# B&R Automation Studio project OpcUaSample410_BrbLibUa103 (part 18)

#### ClientST.st - Implementation code
```iecst
PROGRAM _INIT
	// Initialisierung des Tasks
	brsmemset(ADR(ClientVarsSubscription), 0, SIZEOF(ClientVarsSubscription)); // Auf diese Variablen werden die vom Server geschickten Werte geschrieben
	fbTrigger.PT := T#1s;
	brsmemset(ADR(ClientVarsRead), 0, SIZEOF(ClientVarsRead)); // Auf diese Variablen werden die vom Server gelesenen Werte geschrieben
	brsmemset(ADR(ReceivedEvent), 0, SIZEOF(ReceivedEvent)); // Auf diese Variablen werden die vom Server empfangenen Event-Felder geschrieben

	// Initialisierung der Schrittkette
	Step.eStepNr := eSTEP_INIT;
	bStartClient := 1; // Der Client startet erst, wenn auf 1. Kann zum Debugging auf 0 gesetzt werden.

	// Vorbesetzen der Konfiguration
	ClientCfg.Connection.sServerEndpointUrl := 'opc.tcp://localhost:4840';
	//ClientCfg.Connection.sServerEndpointUrl := 'opc.tcp://192.168.178.37:4840'; // Nur zum Test
	ClientCfg.Connection.UserIdentityToken.UserIdentityTokenType := UAUITT_Username;
	ClientCfg.Connection.UserIdentityToken.TokenParam1 := 'Admin';
	ClientCfg.Connection.UserIdentityToken.TokenParam2 := 'admin';
	ClientCfg.Connection.tSessionTimeout := T#30s;
	ClientCfg.Connection.tMonitorConnection := T#1s;

	ClientCfg.Subscriptions.sNamespaceUriOrg := 'http://opcfoundation.org/UA/'; // NamespaceUri für den Namespace der Foundation
	//ClientCfg.Subscriptions.sNamespaceUriBrPv := 'urn:B&R/pv/'; // NamespaceUri für B&R V1.0
	ClientCfg.Subscriptions.sNamespaceUriBrPv := 'http://br-automation.com/OpcUa/PLC/PV/'; // NamespaceUri für B&R V2.0

	nSubscriptionIndex := 0;
	ClientCfg.Subscriptions.SubVar[nSubscriptionIndex].tPublishingInterval := T#500ms;
	ClientCfg.Subscriptions.SubVar[nSubscriptionIndex].nPriority := 200; // 0..255: Je größer, desto höher die Priorität
	ClientCfg.Subscriptions.SubVar[nSubscriptionIndex].MonitoredItem[0].NodeId.Identifier := '::ServerData:VarsLocal.ReadOnly.bBool';
	ClientCfg.Subscriptions.SubVar[nSubscriptionIndex].MonitoredItem[0].sVarName := '::ClientST:ClientVarsSubscription.bBool';
	ClientCfg.Subscriptions.SubVar[nSubscriptionIndex].MonitoredItem[1].NodeId.Identifier := '::ServerData:VarsLocal.ReadOnly.nUsint';
	ClientCfg.Subscriptions.SubVar[nSubscriptionIndex].MonitoredItem[1].sVarName := '::ClientST:ClientVarsSubscription.nUsint';
	ClientCfg.Subscriptions.SubVar[nSubscriptionIndex].MonitoredItem[2].NodeId.Identifier := '::ServerData:VarsLocal.ReadOnly.nUint';
	ClientCfg.Subscriptions.SubVar[nSubscriptionIndex].MonitoredItem[2].sVarName := '::ClientST:ClientVarsSubscription.nUint';
	ClientCfg.Subscriptions.SubVar[nSubscriptionIndex].MonitoredItem[3].NodeId.Identifier := '::ServerData:VarsLocal.ReadOnly.nUdint';
	ClientCfg.Subscriptions.SubVar[nSubscriptionIndex].MonitoredItem[3].sVarName := '::ClientST:ClientVarsSubscription.nUdint';

	nSubscriptionIndex := 1;
	ClientCfg.Subscriptions.SubVar[nSubscriptionIndex].tPublishingInterval := T#1s;
	ClientCfg.Subscriptions.SubVar[nSubscriptionIndex].nPriority := 100; // 0..255: Je größer, desto höher die Priorität
	ClientCfg.Subscriptions.SubVar[nSubscriptionIndex].MonitoredItem[0].NodeId.Identifier := '::ServerData:VarsLocal.ReadOnly.nSint';
	ClientCfg.Subscriptions.SubVar[nSubscriptionIndex].MonitoredItem[0].sVarName := '::ClientST:ClientVarsSubscription.nSint';
	ClientCfg.Subscriptions.SubVar[nSubscriptionIndex].MonitoredItem[1].NodeId.Identifier := '::ServerData:VarsLocal.ReadOnly.nInt';
	ClientCfg.Subscriptions.SubVar[nSubscriptionIndex].MonitoredItem[1].sVarName := '::ClientST:ClientVarsSubscription.nInt';
	ClientCfg.Subscriptions.SubVar[nSubscriptionIndex].MonitoredItem[2].NodeId.Identifier := '::ServerData:VarsLocal.ReadOnly.nDint';
	ClientCfg.Subscriptions.SubVar[nSubscriptionIndex].MonitoredItem[2].sVarName := '::ClientST:ClientVarsSubscription.nDint';
	ClientCfg.Subscriptions.SubVar[nSubscriptionIndex].MonitoredItem[3].NodeId.Identifier := '::ServerData:VarsLocal.ReadOnly.rReal';
	ClientCfg.Subscriptions.SubVar[nSubscriptionIndex].MonitoredItem[3].sVarName := '::ClientST:ClientVarsSubscription.rReal';

	nSubscriptionIndex := 2;
	ClientCfg.Subscriptions.SubVar[nSubscriptionIndex].tPublishingInterval := T#2s;
	ClientCfg.Subscriptions.SubVar[nSubscriptionIndex].nPriority := 50; // 0..255: Je größer, desto höher die Priorität
	ClientCfg.Subscriptions.SubVar[nSubscriptionIndex].MonitoredItem[0].NodeId.Identifier := '::ServerData:VarsLocal.ReadOnly.rLongReal';
	ClientCfg.Subscriptions.SubVar[nSubscriptionIndex].MonitoredItem[0].sVarName := '::ClientST:ClientVarsSubscription.rLongReal';
	ClientCfg.Subscriptions.SubVar[nSubscriptionIndex].MonitoredItem[1].NodeId.Identifier := '::ServerData:VarsLocal.ReadOnly.sString';
	ClientCfg.Subscriptions.SubVar[nSubscriptionIndex].MonitoredItem[1].sVarName := '::ClientST:ClientVarsSubscription.sString';
	ClientCfg.Subscriptions.SubVar[nSubscriptionIndex].MonitoredItem[2].NodeId.Identifier := '::ServerData:VarsLocal.ReadOnly.tTime';
	ClientCfg.Subscriptions.SubVar[nSubscriptionIndex].MonitoredItem[2].sVarName := '::ClientST:ClientVarsSubscription.tTime';
	ClientCfg.Subscriptions.SubVar[nSubscriptionIndex].MonitoredItem[3].NodeId.Identifier := '::ServerData:VarsLocal.ReadOnly.dtDateTime';
	ClientCfg.Subscriptions.SubVar[nSubscriptionIndex].MonitoredItem[3].sVarName := '::ClientST:ClientVarsSubscription.dtDateTime';

	MonitoredItemParameter.SamplingInterval := 0; // Wird von Subscription.PublishingInterval abgeleitet
	MonitoredItemParameter.QueueSize := 0; // Wenn > 0, dann müsste zyklisch der FB 'UA_MonitoredItemOperateList' für jede Subscription ausgeführt werden
	MonitoredItemParameter.DiscardOldest := 1;
	MonitoredItemParameter.DeadbandType := UADeadbandType_None;
	MonitoredItemParameter.Deadband := 0.0;
	FOR nSubscriptionIndex := 0 TO nCLIENT_SUBSCRIPTION_INDEX_MAX DO
		FOR nItemIndex := 0 TO nCLIENT_MONITORED_ITEM_INDEX_MAX DO
			ClientCfg.Subscriptions.SubVar[nSubscriptionIndex].MonitoredItem[nItemIndex].NodeId.NamespaceIndex := 0; // Der NamespaceIndex wird später einmalig ermiitelt und dann zugewiesen
			ClientCfg.Subscriptions.SubVar[nSubscriptionIndex].MonitoredItem[nItemIndex].NodeId.IdentifierType := UAIdentifierType_String;
		END_FOR
	END_FOR

	ClientCfg.Subscriptions.SubEvt.tPublishingInterval := t#100ms;
	ClientCfg.Subscriptions.SubEvt.nPriority := 250; // 0..255: Je größer, desto höher die Priorität
	ClientCfg.Subscriptions.SubEvt.NotifierNodeId.IdentifierType := UAIdentifierType_Numeric;
	ClientCfg.Subscriptions.SubEvt.NotifierNodeId.Identifier := '2253'; // Root/Objects/Server
	ClientCfg.Subscriptions.SubEvt.EventTypeNodeId.IdentifierType := UAIdentifierType_Numeric;
	ClientCfg.Subscriptions.SubEvt.EventTypeNodeId.Identifier := '11436'; // Root/Types/EventTypes/BaseEventType/ProgressEventType

	brsmemset(ADR(asReadVars), 0, SIZEOF(asReadVars));
	ClientCfg.Read.Item[0].NodeId.Identifier := '::ServerData:VarsLocal.ReadOnly.nUdint';
	ClientCfg.Read.Item[0].sVarName := '::ClientST:ClientVarsRead.nUdint';
	ClientCfg.Read.Item[1].NodeId.Identifier := '::ServerData:VarsLocal.ReadOnly.nDint';
	ClientCfg.Read.Item[1].sVarName := '::ClientST:ClientVarsRead.nDint';
	ClientCfg.Read.Item[2].NodeId.Identifier := '::ServerData:VarsLocal.ReadOnly.anInt';
	ClientCfg.Read.Item[2].sVarName := '::ClientST:ClientVarsRead.anInt';
	FOR nItemIndex := 0 TO nCLIENT_READ_ITEM_INDEX_MAX DO
		ClientCfg.Read.Item[nItemIndex].NodeId.NamespaceIndex := 0; // Der NamespaceIndex wird später einmalig ermiitelt und dann zugewiesen
		ClientCfg.Read.Item[nItemIndex].NodeId.IdentifierType := UAIdentifierType_String;
	END_FOR

	brsmemset(ADR(asWriteVars), 0, SIZEOF(asWriteVars));
	ClientCfg.Write.Item[0].NodeId.Identifier := '::ServerData:WriteST.nUdint';
	ClientCfg.Write.Item[0].sVarName := '::ClientST:ClientVarsRead.nUdint';
	ClientCfg.Write.Item[1].NodeId.Identifier := '::ServerData:WriteST.nDint';
	ClientCfg.Write.Item[1].sVarName := '::ClientST:ClientVarsRead.nDint';
	ClientCfg.Write.Item[2].NodeId.Identifier := '::ServerData:WriteST.anInt';
	ClientCfg.Write.Item[2].sVarName := '::ClientST:ClientVarsRead.anInt';
	FOR nItemIndex := 0 TO nCLIENT_WRITE_ITEM_INDEX_MAX DO
		ClientCfg.Write.Item[nItemIndex].NodeId.NamespaceIndex := 0; // Der NamespaceIndex wird später einmalig ermiitelt und dann zugewiesen
		ClientCfg.Write.Item[nItemIndex].NodeId.IdentifierType := UAIdentifierType_String;
	END_FOR

	brsmemset(ADR(MethCalculateArgs), 0, SIZEOF(MethCalculateArgs));
	ClientCfg.Methods.Method[0].ObjectNodeId.Identifier := '::SrvMethST'; // Task-Node
	ClientCfg.Methods.Method[0].MethodNodeId.Identifier := '::SrvMethST:Calculate'; // Method-Node
	ClientCfg.Methods.Method[0].ArgumentsIn[0].Name := 'nValue0'; // Name des Eingans wie in der Methode deklariert
	ClientCfg.Methods.Method[0].ArgumentsIn[0].Value := '::ClientST:MethCalculateArgs.In.nVal0'; // Name der Variable, auf die der Wert des Eingang geschrieben wird
	ClientCfg.Methods.Method[0].ArgumentsIn[1].Name := 'nValue1';
	ClientCfg.Methods.Method[0].ArgumentsIn[1].Value := '::ClientST:MethCalculateArgs.In.nVal1';
	ClientCfg.Methods.Method[0].ArgumentsIn[2].Name := 'anArrayIn';
	ClientCfg.Methods.Method[0].ArgumentsIn[2].Value := '::ClientST:MethCalculateArgs.In.anArray';
	ClientCfg.Methods.Method[0].ArgumentsOut[0].Name := 'nAddition'; // Name des Ausgangs wie in der Methode deklariert
	ClientCfg.Methods.Method[0].ArgumentsOut[0].Value := '::ClientST:MethCalculateArgs.Out.nAddition'; // Name der Variable, von der der Wert des Ausgangs genommen wird
	ClientCfg.Methods.Method[0].ArgumentsOut[1].Name := 'nMultiplication';
	ClientCfg.Methods.Method[0].ArgumentsOut[1].Value := '::ClientST:MethCalculateArgs.Out.nMultiplication';
	ClientCfg.Methods.Method[0].ArgumentsOut[2].Name := 'anArrayOut';
	ClientCfg.Methods.Method[0].ArgumentsOut[2].Value := '::ClientST:MethCalculateArgs.Out.anArray';
	FOR nItemIndex := 0 TO nCLIENT_METHODS_INDEX_MAX DO
		ClientCfg.Methods.Method[0].ObjectNodeId.NamespaceIndex := 0; // Der NamespaceIndex wird später einmalig ermiitelt und dann zugewiesen
		ClientCfg.Methods.Method[0].ObjectNodeId.IdentifierType := UAIdentifierType_String;
		ClientCfg.Methods.Method[0].MethodNodeId.NamespaceIndex := 0; // Der NamespaceIndex wird später einmalig ermiitelt und dann zugewiesen
		ClientCfg.Methods.Method[0].MethodNodeId.IdentifierType := UAIdentifierType_String;
	END_FOR

	// Ablöschen der Funktionsblöcke und Strukturen
	brsmemset(ADR(fbUA_ConnectionGetStatus), 0, SIZEOF(fbUA_ConnectionGetStatus));
	brsmemset(ADR(fbUA_Connect), 0, SIZEOF(fbUA_Connect));
	brsmemset(ADR(fbUA_Disconnect), 0, SIZEOF(fbUA_Disconnect));
	brsmemset(ADR(fbUA_GetNamespaceIndex), 0, SIZEOF(fbUA_GetNamespaceIndex));
	brsmemset(ADR(fbUA_SubscriptionCreate), 0, SIZEOF(fbUA_SubscriptionCreate));
	brsmemset(ADR(fbUA_NodeGetHandleList), 0, SIZEOF(fbUA_NodeGetHandleList));
	brsmemset(ADR(fbUA_MonitoredItemAddList), 0, SIZEOF(fbUA_MonitoredItemAddList));
	brsmemset(ADR(fbUA_MethodGetHandle), 0, SIZEOF(fbUA_MethodGetHandle));
	brsmemset(ADR(fbUA_ReadList), 0, SIZEOF(fbUA_ReadList));
	brsmemset(ADR(fbUA_WriteList), 0, SIZEOF(fbUA_WriteList));
	brsmemset(ADR(fbUA_MethodCall), 0, SIZEOF(fbUA_MethodCall));
END_PROGRAM

PROGRAM _CYCLIC
	// Schrittkette
	CASE Step.eStepNr OF
		eSTEP_NONE:

		eSTEP_INIT:
			IF bStartClient = 1 THEN
				Step.eStepNr := eSTEP_CONNECT;
			END_IF

		// -----------------------------------------------------------------------------------------------------------------------------------------------
		eSTEP_CONNECT:
			// Hier wird die Verbindung zum Server aufgebaut.
			brsmemset(ADR(fbUA_Connect), 0, SIZEOF(fbUA_Connect));
			fbUA_Connect.Execute := 1;
			fbUA_Connect.ServerEndpointUrl := ClientCfg.Connection.sServerEndpointUrl;
			fbUA_Connect.SessionConnectInfo.SessionName := 'SampleClientST_Session';
			fbUA_Connect.SessionConnectInfo.ApplicationName := 'SampleClientST_Application';
			fbUA_Connect.SessionConnectInfo.SecurityMsgMode := UASecurityMsgMode_None; // Ohne Security
			fbUA_Connect.SessionConnectInfo.SecurityPolicy := UASecurityPolicy_None; // Ohne Security
			fbUA_Connect.SessionConnectInfo.CertificateStore := 'SslCfgOpcUaClient'; // // Angabe der SSL-Configuration unter 'ConfigurationView/AccessAndSecurity/TransortLayerSecurity/OpcUaCfg.sslcfg'
			fbUA_Connect.SessionConnectInfo.ClientCertificateName := ''; // Muss leer bleiben
			fbUA_Connect.SessionConnectInfo.ServerUri := ''; // Kann leer bleiben
			fbUA_Connect.SessionConnectInfo.CheckServerCertificate := 0;
			fbUA_Connect.SessionConnectInfo.TransportProfile := UATP_UATcp;
			brsmemcpy(ADR(fbUA_Connect.SessionConnectInfo.UserIdentityToken), ADR(ClientCfg.Connection.UserIdentityToken), SIZEOF(UAUserIdentityToken));
			fbUA_Connect.SessionConnectInfo.VendorSpecificParameter := ''; // Kann leer bleiben
			fbUA_Connect.SessionConnectInfo.SessionTimeout := ClientCfg.Connection.tSessionTimeout;
			fbUA_Connect.SessionConnectInfo.MonitorConnection := ClientCfg.Connection.tMonitorConnection;
			fbUA_Connect.SessionConnectInfo.LocaleIDs[0] := 'de';
			fbUA_Connect.Timeout := tFB_TIMEOUT;
			nConnectionHandle := 0;
			Step.eStepNr := eSTEP_CONNECT_WAIT;

		eSTEP_CONNECT_WAIT:
			// Aufruf abwarten
			IF fbUA_Connect.Busy = 0 THEN
				fbUA_Connect.Execute := 0;
				IF fbUA_Connect.Done = 1 THEN
					nConnectionHandle := fbUA_Connect.ConnectionHdl;
					Step.eStepNr := eSTEP_GET_NAMESPACEIDX_ORG;
				ELSIF fbUA_Connect.Error = 1 THEN
						// Ständig versuchen, die Verbindung aufzubauen
						nConnectionHandle := 0;
						Step.eStepNr := eSTEP_CONNECT;
				END_IF
			END_IF

		// -----------------------------------------------------------------------------------------------------------------------------------------------
		eSTEP_GET_NAMESPACEIDX_ORG:
			// Hier wird der Namespace-Uri vom Server in einen Index übersetzt (für den Namespace der Foundation)
			brsmemset(ADR(fbUA_GetNamespaceIndex), 0, SIZEOF(fbUA_GetNamespaceIndex));
			fbUA_GetNamespaceIndex.Execute := 1;
			fbUA_GetNamespaceIndex.ConnectionHdl := nConnectionHandle;
			fbUA_GetNamespaceIndex.NamespaceUri := ClientCfg.Subscriptions.sNamespaceUriOrg;
			fbUA_GetNamespaceIndex.Timeout := tFB_TIMEOUT;
			Step.eStepNr := eSTEP_GET_NAMESPACEIDX_ORG_WAIT;

		eSTEP_GET_NAMESPACEIDX_ORG_WAIT:
			// Aufruf abwarten
			IF fbUA_GetNamespaceIndex.Busy = 0 THEN
				fbUA_GetNamespaceIndex.Execute := 0;
				IF fbUA_GetNamespaceIndex.Done = 1 THEN
					ClientCfg.Subscriptions.nNamespaceUriOrg := fbUA_GetNamespaceIndex.NamespaceIndex;
					ClientCfg.Subscriptions.SubEvt.NotifierNodeId.NamespaceIndex := ClientCfg.Subscriptions.nNamespaceUriOrg;
					ClientCfg.Subscriptions.SubEvt.EventTypeNodeId.NamespaceIndex := ClientCfg.Subscriptions.nNamespaceUriOrg;
					Step.eStepNr := eSTEP_GET_NAMESPACEIDX_BRPV;
				ELSIF fbUA_GetNamespaceIndex.Error = 1 THEN
					Step.eErrorStep := Step.eStepNr;
					Step.nSubscriptionIndex := -1;
					Step.nItemIndex := -1;
					Step.nErrorId := fbUA_GetNamespaceIndex.ErrorID;
					Step.eStepNr := eSTEP_PAR_ERROR;
				END_IF
			END_IF

		eSTEP_GET_NAMESPACEIDX_BRPV:
			// Hier wird der Namespace-Uri vom Server in einen Index übersetzt.	Bei B&R-PV ist nur ein Namespace benötigt.
			brsmemset(ADR(fbUA_GetNamespaceIndex), 0, SIZEOF(fbUA_GetNamespaceIndex));
			fbUA_GetNamespaceIndex.Execute := 1;
			fbUA_GetNamespaceIndex.ConnectionHdl := nConnectionHandle;
			fbUA_GetNamespaceIndex.NamespaceUri := ClientCfg.Subscriptions.sNamespaceUriBrPv;
			fbUA_GetNamespaceIndex.Timeout := tFB_TIMEOUT;
			Step.eStepNr := eSTEP_GET_NAMESPACEIDX_BRPV_WAIT;

		eSTEP_GET_NAMESPACEIDX_BRPV_WAIT:
			// Aufruf abwarten
			IF fbUA_GetNamespaceIndex.Busy = 0 THEN
				fbUA_GetNamespaceIndex.Execute := 0;
				IF fbUA_GetNamespaceIndex.Done = 1 THEN
					ClientCfg.Subscriptions.nNamespaceUriBrPv := fbUA_GetNamespaceIndex.NamespaceIndex;
					// NamespaceIndex auf alle MonitoredItems übernehmen
					FOR nSubscriptionIndex := 0 TO nCLIENT_SUBSCRIPTION_INDEX_MAX DO
						FOR nItemIndex := 0 TO nCLIENT_MONITORED_ITEM_INDEX_MAX DO
							ClientCfg.Subscriptions.SubVar[nSubscriptionIndex].MonitoredItem[nItemIndex].NodeId.NamespaceIndex := fbUA_GetNamespaceIndex.NamespaceIndex;
						END_FOR
					END_FOR
					// NamespaceIndex auf alle ReadItems übernehmen
					FOR nItemIndex := 0 TO nCLIENT_READ_ITEM_INDEX_MAX DO
						ClientCfg.Read.Item[nItemIndex].NodeId.NamespaceIndex := fbUA_GetNamespaceIndex.NamespaceIndex;
					END_FOR
					// NamespaceIndex auf alle WriteItems übernehmen
					FOR nItemIndex := 0 TO nCLIENT_WRITE_ITEM_INDEX_MAX DO
						ClientCfg.Write.Item[nItemIndex].NodeId.NamespaceIndex := fbUA_GetNamespaceIndex.NamespaceIndex;
					END_FOR
					// NamespaceIndex auf alle Methods übernehmen
					FOR nItemIndex := 0 TO nCLIENT_METHODS_INDEX_MAX DO
						ClientCfg.Methods.Method[nItemIndex].MethodNodeId.NamespaceIndex := fbUA_GetNamespaceIndex.NamespaceIndex;
						ClientCfg.Methods.Method[nItemIndex].ObjectNodeId.NamespaceIndex := fbUA_GetNamespaceIndex.NamespaceIndex;
					END_FOR
					Step.eStepNr := eSTEP_CREATE_SUBSCRIPTIONS_VAR;
				ELSIF fbUA_GetNamespaceIndex.Error = 1 THEN
					Step.eErrorStep := Step.eStepNr;
					Step.nSubscriptionIndex := -1;
					Step.nItemIndex := -1;
					Step.nErrorId := fbUA_GetNamespaceIndex.ErrorID;
					Step.eStepNr := eSTEP_PAR_ERROR;
				END_IF
			END_IF

			// -----------------------------------------------------------------------------------------------------------------------------------------------
		eSTEP_CREATE_SUBSCRIPTIONS_VAR:
			nSubscriptionIndex := -1; // Mit der ersten Subscription beginnen
			Step.eStepNr := eSTEP_CREATE_SUBSCRIPTION_VAR;

		eSTEP_CREATE_SUBSCRIPTION_VAR:
			// Nächste Subscription hinzufügen
			nSubscriptionIndex := nSubscriptionIndex + 1;
			IF nSubscriptionIndex <= nCLIENT_SUBSCRIPTION_INDEX_MAX THEN
				// Nächste Subscription anlegen
				brsmemset(ADR(fbUA_SubscriptionCreate), 0, SIZEOF(fbUA_SubscriptionCreate));
				fbUA_SubscriptionCreate.Execute := 1;
				fbUA_SubscriptionCreate.ConnectionHdl := nConnectionHandle;
				fbUA_SubscriptionCreate.PublishingEnable := 1;
				fbUA_SubscriptionCreate.Priority := ClientCfg.Subscriptions.SubVar[nSubscriptionIndex].nPriority;
				fbUA_SubscriptionCreate.Timeout := tFB_TIMEOUT;
				// Unter ST können IN/OUT-Elemente nicht direkt angegeben werden, sondern nur beim FB-Aufruf (siehe unten)
				tSubscriptionPublishingInterval := ClientCfg.Subscriptions.SubVar[nSubscriptionIndex].tPublishingInterval;
				Step.eStepNr := eSTEP_CREATE_SUBSCRIPT_VAR_WAIT;
			ELSE
				// Alle Subscriptions angelegt
				IF Step.nErrorId <> 0 THEN
					Step.eStepNr := eSTEP_PAR_ERROR;
				ELSE
					Step.eStepNr := eSTEP_CREATE_SUBSCRIPTION_EVT;
				END_IF
			END_IF

		eSTEP_CREATE_SUBSCRIPT_VAR_WAIT:
			// Aufruf abwarten
			IF fbUA_SubscriptionCreate.Busy = 0 THEN
				fbUA_SubscriptionCreate.Execute := 0;
				IF fbUA_SubscriptionCreate.Done = 1 THEN
					Step.eStepNr := eSTEP_SUB_GET_NODE_HDL_LIST;
				ELSIF fbUA_SubscriptionCreate.Error = 1 THEN
					// Fehler eintragen, aber trotzdem mit der nächsten Subcription weiter machen
					Step.eErrorStep := Step.eStepNr;
					Step.nSubscriptionIndex := nSubscriptionIndex;
					Step.nItemIndex := -1;
					Step.nErrorId := fbUA_SubscriptionCreate.ErrorID;
					Step.eStepNr := eSTEP_CREATE_SUBSCRIPTION_VAR;
				END_IF
			END_IF

		eSTEP_SUB_GET_NODE_HDL_LIST:
			// Die Handles für die MonitoredItems ermitteln
			brsmemset(ADR(fbUA_NodeGetHandleList), 0, SIZEOF(fbUA_NodeGetHandleList));
			fbUA_NodeGetHandleList.Execute := 1;
			fbUA_NodeGetHandleList.ConnectionHdl := nConnectionHandle;
			FOR nItemIndex := 0 TO nCLIENT_MONITORED_ITEM_INDEX_MAX DO
				IF brsstrlen(ADR(ClientCfg.Subscriptions.SubVar[nSubscriptionIndex].MonitoredItem[nItemIndex].NodeId.Identifier)) > 0 THEN
					brsmemcpy(ADR(fbUA_NodeGetHandleList.NodeIDs[nItemIndex]), ADR(ClientCfg.Subscriptions.SubVar[nSubscriptionIndex].MonitoredItem[nItemIndex].NodeId), SIZEOF(UANodeID));
				ELSE
					EXIT;
				END_IF
			END_FOR
			fbUA_NodeGetHandleList.NodeIDCount := nItemIndex;
			fbUA_NodeGetHandleList.Timeout := tFB_TIMEOUT;
			Step.eStepNr := eSTEP_SUB_GET_NODE_HDL_LIST_WAIT;

		eSTEP_SUB_GET_NODE_HDL_LIST_WAIT:
			// Aufruf abwarten
			IF fbUA_NodeGetHandleList.Busy = 0 THEN
				fbUA_NodeGetHandleList.Execute := 0;
				IF fbUA_NodeGetHandleList.Done = 1 THEN
					nItemIndex := -1;
					Step.eStepNr := eSTEP_ADD_MONITORED_ITEMS;
				ELSIF fbUA_NodeGetHandleList.Error = 1 THEN
					// Fehler eintragen, aber trotzdem weiter machen
					Step.eErrorStep := Step.eStepNr;
					Step.nSubscriptionIndex := nSubscriptionIndex;
					IF fbUA_NodeGetHandleList.ErrorID <> 0 THEN
						Step.nItemIndex := -1;
						Step.nErrorId := fbUA_NodeGetHandleList.ErrorID;
					ELSE
						FOR nItemIndex := 0 TO MAX_INDEX_NODELIST DO
							IF fbUA_NodeGetHandleList.NodeErrorIDs[nItemIndex] <> 0 THEN
								Step.nItemIndex := nItemIndex;
								Step.nErrorId := fbUA_NodeGetHandleList.NodeErrorIDs[nItemIndex];
								EXIT;
							END_IF
						END_FOR
					END_IF
					nItemIndex := -1;
					Step.eStepNr := eSTEP_CREATE_SUBSCRIPTION_VAR;
				END_IF
			END_IF

		eSTEP_ADD_MONITORED_ITEMS:
			// MonitoredItems hinzufügen
			brsmemset(ADR(fbUA_MonitoredItemAddList), 0, SIZEOF(fbUA_MonitoredItemAddList));
			fbUA_MonitoredItemAddList.Execute := 1;
			fbUA_MonitoredItemAddList.SubscriptionHdl := fbUA_SubscriptionCreate.SubscriptionHdl;
			FOR nItemIndex := 0 TO nCLIENT_MONITORED_ITEM_INDEX_MAX DO
				IF brsstrlen(ADR(ClientCfg.Subscriptions.SubVar[nSubscriptionIndex].MonitoredItem[nItemIndex].NodeId.Identifier)) > 0 THEN
					fbUA_MonitoredItemAddList.NodeHdls[nItemIndex] := fbUA_NodeGetHandleList.NodeHdls[nItemIndex];
					fbUA_MonitoredItemAddList.NodeAddInfos[nItemIndex].AttributeId := UAAI_Value; // Es ist möglich, alle Attribute eines Nodes zu adressieren, aber normalerweise wird natürlich das Attribut 'Value' benötigt
					fbUA_MonitoredItemAddList.NodeAddInfos[nItemIndex].IndexRangeCount := 0; // Nur Einzel-Variablen, keine Arrays
					brsmemset(ADR(fbUA_MonitoredItemAddList.NodeAddInfos[nItemIndex].IndexRange), 0, SIZEOF(fbUA_MonitoredItemAddList.NodeAddInfos[nItemIndex].IndexRange));
					asMonitoredItemVarNames[nItemIndex] := ClientCfg.Subscriptions.SubVar[nSubscriptionIndex].MonitoredItem[nItemIndex].sVarName;
					brsmemcpy(ADR(aMonitoredItemParameter[nItemIndex]), ADR(MonitoredItemParameter), SIZEOF(MonitoredItemParameter));
					aMonitoredItemParameter[nItemIndex].SamplingInterval := ClientCfg.Subscriptions.SubVar[nSubscriptionIndex].tPublishingInterval; // Nur das SamplingInterval wird von der Subscription abgeleitet
				ELSE
					EXIT;
				END_IF
			END_FOR
			fbUA_MonitoredItemAddList.NodeHdlCount := nItemIndex;
			fbUA_MonitoredItemAddList.Timeout := tFB_TIMEOUT;
			// Unter ST können IN/OUT-Elemente nicht direkt angegeben werden, sondern nur beim FB-Aufruf (siehe unten)
			Step.eStepNr := eSTEP_ADD_MONITORED_ITEMS_WAIT;

		eSTEP_ADD_MONITORED_ITEMS_WAIT:
			// Aufruf abwarten
			IF fbUA_MonitoredItemAddList.Busy = 0 THEN
				fbUA_MonitoredItemAddList.Execute := 0;
				IF fbUA_MonitoredItemAddList.Done = 1 THEN
					Step.eStepNr := eSTEP_CREATE_SUBSCRIPTION_VAR;
				ELSIF fbUA_MonitoredItemAddList.Error = 1 THEN
					// Fehler eintragen, aber trotzdem weiter machen
					Step.eErrorStep := Step.eStepNr;
					Step.nSubscriptionIndex := nSubscriptionIndex;
					IF fbUA_MonitoredItemAddList.ErrorID <> 0 THEN
						Step.nItemIndex := -1;
						Step.nErrorId := fbUA_MonitoredItemAddList.ErrorID;
					ELSE
						FOR nItemIndex := 0 TO MAX_INDEX_NODELIST DO
							IF fbUA_MonitoredItemAddList.NodeErrorIDs[nItemIndex] <> 0 THEN
								Step.nItemIndex := nItemIndex;
								Step.nErrorId := fbUA_MonitoredItemAddList.NodeErrorIDs[nItemIndex];
								EXIT;
							END_IF
						END_FOR
					END_IF
					Step.eStepNr := eSTEP_CREATE_SUBSCRIPTION_VAR;
				END_IF
			END_IF

		// -----------------------------------------------------------------------------------------------------------------------------------------------
		eSTEP_CREATE_SUBSCRIPTION_EVT:
			// Subscription für Event hinzufügen
			brsmemset(ADR(fbUA_SubscriptionCreate), 0, SIZEOF(fbUA_SubscriptionCreate));
			fbUA_SubscriptionCreate.Execute := 1;
			fbUA_SubscriptionCreate.ConnectionHdl := nConnectionHandle;
			fbUA_SubscriptionCreate.PublishingEnable := 1;
			fbUA_SubscriptionCreate.Priority := ClientCfg.Subscriptions.SubEvt.nPriority;
			fbUA_SubscriptionCreate.Timeout := tFB_TIMEOUT;
			tSubscriptionPublishingInterval := ClientCfg.Subscriptions.SubEvt.tPublishingInterval;
			Step.eStepNr := eSTEP_CREATE_SUBSCRIPT_EVT_WAIT;

		eSTEP_CREATE_SUBSCRIPT_EVT_WAIT:
			// Aufruf abwarten
			IF fbUA_SubscriptionCreate.Busy = 0 THEN
				fbUA_SubscriptionCreate.Execute := 0;
				IF fbUA_SubscriptionCreate.Done = 1 THEN
					Step.eStepNr := eSTEP_EVT_GET_NODE_HDL;
				ELSIF fbUA_SubscriptionCreate.Error = 1 THEN
					// Fehler eintragen, aber trotzdem weiter machen
					Step.eErrorStep := Step.eStepNr;
					Step.nSubscriptionIndex := -1;
					Step.nItemIndex := -1;
					Step.nErrorId := fbUA_SubscriptionCreate.ErrorID;
					Step.eStepNr := eSTEP_RD_GET_NODE_HDL_LIST;
				END_IF
			END_IF

		eSTEP_EVT_GET_NODE_HDL:
			brsmemset(ADR(fbUA_NodeGetHandle), 0, SIZEOF(fbUA_NodeGetHandle));
			fbUA_NodeGetHandle.Execute := 1;
			fbUA_NodeGetHandle.ConnectionHdl := nConnectionHandle;
			brsmemcpy(ADR(fbUA_NodeGetHandle.NodeID), ADR(ClientCfg.Subscriptions.SubEvt.NotifierNodeId), SIZEOF(UANodeID)); // Root/Objects/Server
			fbUA_NodeGetHandle.Timeout := tFB_TIMEOUT;
			Step.eStepNr := eSTEP_EVT_GET_NODE_HDL_WAIT;

		eSTEP_EVT_GET_NODE_HDL_WAIT:
			// Aufruf abwarten
			IF fbUA_NodeGetHandle.Busy = 0 THEN
				fbUA_NodeGetHandle.Execute := 0;
				IF fbUA_NodeGetHandle.Done = 1 THEN
					Step.eStepNr := eSTEP_ADD_EVENT_ITEM;
				ELSIF fbUA_NodeGetHandle.Error = 1 THEN
					// Fehler eintragen, aber trotzdem weiter machen
					Step.eErrorStep := Step.eStepNr;
					Step.nSubscriptionIndex := -1;
					Step.nErrorId := fbUA_NodeGetHandle.ErrorID;
					Step.eStepNr := eSTEP_RD_GET_NODE_HDL_LIST;
				END_IF
			END_IF

		eSTEP_ADD_EVENT_ITEM:
			fbUA_EventItemAdd.Execute := 1;
			fbUA_EventItemAdd.SubscriptionHdl := fbUA_SubscriptionCreate.SubscriptionHdl;
			fbUA_EventItemAdd.NodeHdl := fbUA_NodeGetHandle.NodeHdl; // Root/Objects/Server
			// Event-Typ festlegen
			brsmemcpy(ADR(fbUA_EventItemAdd.EventType), ADR(ClientCfg.Subscriptions.SubEvt.EventTypeNodeId), SIZEOF(UANodeID));
			// Zu sendende Felder festlegen
			// EventId
			nItemIndex := 0;
			fbUA_EventItemAdd.EventFieldSelections[nItemIndex].NoOfElements := 1;
			fbUA_EventItemAdd.EventFieldSelections[nItemIndex].Elements[0].TargetName.NamespaceIndex := ClientCfg.Subscriptions.nNamespaceUriOrg;
			fbUA_EventItemAdd.EventFieldSelections[nItemIndex].Elements[0].TargetName.Name := 'EventId';
			ClientCfg.Subscriptions.SubEvt.EventFieldVarNames[nItemIndex] := '::ClientST:ReceivedEvent.EventId';
			// EventType
			nItemIndex := nItemIndex + 1;
			fbUA_EventItemAdd.EventFieldSelections[nItemIndex].NoOfElements := 1;
			fbUA_EventItemAdd.EventFieldSelections[nItemIndex].Elements[0].TargetName.NamespaceIndex := ClientCfg.Subscriptions.nNamespaceUriOrg;
			fbUA_EventItemAdd.EventFieldSelections[nItemIndex].Elements[0].TargetName.Name := 'EventType';
			ClientCfg.Subscriptions.SubEvt.EventFieldVarNames[nItemIndex] := '::ClientST:ReceivedEvent.EventType';
			// LocalTime
			nItemIndex := nItemIndex + 1;
			fbUA_EventItemAdd.EventFieldSelections[nItemIndex].NoOfElements := 1;
			fbUA_EventItemAdd.EventFieldSelections[nItemIndex].Elements[0].TargetName.NamespaceIndex := ClientCfg.Subscriptions.nNamespaceUriOrg;
			fbUA_EventItemAdd.EventFieldSelections[nItemIndex].Elements[0].TargetName.Name := 'LocalTime';
			ClientCfg.Subscriptions.SubEvt.EventFieldVarNames[nItemIndex] := '::ClientST:ReceivedEvent.LocalTime';
			// Message
			nItemIndex := nItemIndex + 1;
			fbUA_EventItemAdd.EventFieldSelections[nItemIndex].NoOfElements := 1;
			fbUA_EventItemAdd.EventFieldSelections[nItemIndex].Elements[0].TargetName.NamespaceIndex := ClientCfg.Subscriptions.nNamespaceUriOrg;
			fbUA_EventItemAdd.EventFieldSelections[nItemIndex].Elements[0].TargetName.Name := 'Message';
			ClientCfg.Subscriptions.SubEvt.EventFieldVarNames[nItemIndex] := '::ClientST:ReceivedEvent.Message';
			// ReceiveTime
			nItemIndex := nItemIndex + 1;
			fbUA_EventItemAdd.EventFieldSelections[nItemIndex].NoOfElements := 1;
			fbUA_EventItemAdd.EventFieldSelections[nItemIndex].Elements[0].TargetName.NamespaceIndex := ClientCfg.Subscriptions.nNamespaceUriOrg;
			fbUA_EventItemAdd.EventFieldSelections[nItemIndex].Elements[0].TargetName.Name := 'ReceiveTime';
			ClientCfg.Subscriptions.SubEvt.EventFieldVarNames[nItemIndex] := '::ClientST:ReceivedEvent.ReceiveTime';
			// Severity
			nItemIndex := nItemIndex + 1;
			fbUA_EventItemAdd.EventFieldSelections[nItemIndex].NoOfElements := 1;
			fbUA_EventItemAdd.EventFieldSelections[nItemIndex].Elements[0].TargetName.NamespaceIndex := ClientCfg.Subscriptions.nNamespaceUriOrg;
			fbUA_EventItemAdd.EventFieldSelections[nItemIndex].Elements[0].TargetName.Name := 'Severity';
			ClientCfg.Subscriptions.SubEvt.EventFieldVarNames[nItemIndex] := '::ClientST:ReceivedEvent.Severity';
			// SourceName
			nItemIndex := nItemIndex + 1;
			fbUA_EventItemAdd.EventFieldSelections[nItemIndex].NoOfElements := 1;
			fbUA_EventItemAdd.EventFieldSelections[nItemIndex].Elements[0].TargetName.NamespaceIndex := ClientCfg.Subscriptions.nNamespaceUriOrg;
			fbUA_EventItemAdd.EventFieldSelections[nItemIndex].Elements[0].TargetName.Name := 'SourceName';
			ClientCfg.Subscriptions.SubEvt.EventFieldVarNames[nItemIndex] := '::ClientST:ReceivedEvent.SourceName';
			// SourceNode
			nItemIndex := nItemIndex + 1;
			fbUA_EventItemAdd.EventFieldSelections[nItemIndex].NoOfElements := 1;
			fbUA_EventItemAdd.EventFieldSelections[nItemIndex].Elements[0].TargetName.NamespaceIndex := ClientCfg.Subscriptions.nNamespaceUriOrg;
			fbUA_EventItemAdd.EventFieldSelections[nItemIndex].Elements[0].TargetName.Name := 'SourceNode';
			ClientCfg.Subscriptions.SubEvt.EventFieldVarNames[nItemIndex] := '::ClientST:ReceivedEvent.SourceNode';
			// Time
			nItemIndex := nItemIndex + 1;
			fbUA_EventItemAdd.EventFieldSelections[nItemIndex].NoOfElements := 1;
			fbUA_EventItemAdd.EventFieldSelections[nItemIndex].Elements[0].TargetName.NamespaceIndex := ClientCfg.Subscriptions.nNamespaceUriOrg;
			fbUA_EventItemAdd.EventFieldSelections[nItemIndex].Elements[0].TargetName.Name := 'Time';
			ClientCfg.Subscriptions.SubEvt.EventFieldVarNames[nItemIndex] := '::ClientST:ReceivedEvent.Time';
			// Context
			nItemIndex := nItemIndex + 1;
			fbUA_EventItemAdd.EventFieldSelections[nItemIndex].NoOfElements := 1;
			fbUA_EventItemAdd.EventFieldSelections[nItemIndex].Elements[0].TargetName.NamespaceIndex := ClientCfg.Subscriptions.nNamespaceUriOrg;
			fbUA_EventItemAdd.EventFieldSelections[nItemIndex].Elements[0].TargetName.Name := 'Context';
			ClientCfg.Subscriptions.SubEvt.EventFieldVarNames[nItemIndex] := '::ClientST:ReceivedEvent.Context';
			// Progress
			nItemIndex := nItemIndex + 1;
			fbUA_EventItemAdd.EventFieldSelections[nItemIndex].NoOfElements := 1;
			fbUA_EventItemAdd.EventFieldSelections[nItemIndex].Elements[0].TargetName.NamespaceIndex := ClientCfg.Subscriptions.nNamespaceUriOrg;
			fbUA_EventItemAdd.EventFieldSelections[nItemIndex].Elements[0].TargetName.Name := 'Progress';
			ClientCfg.Subscriptions.SubEvt.EventFieldVarNames[nItemIndex] := '::ClientST:ReceivedEvent.Progress';
			fbUA_EventItemAdd.EventFieldSelectionCount := nItemIndex + 1;
			fbUA_EventItemAdd.Timeout := tFB_TIMEOUT;
			Step.eStepNr := eSTEP_ADD_EVENT_ITEM_WAIT;

		eSTEP_ADD_EVENT_ITEM_WAIT:
			// Aufruf abwarten
			IF fbUA_EventItemAdd.Busy = 0 THEN
				fbUA_EventItemAdd.Execute := 0;
				IF fbUA_EventItemAdd.Done = 1 THEN
					Step.eStepNr := eSTEP_RD_GET_NODE_HDL_LIST;
				ELSIF fbUA_EventItemAdd.Error = 1 THEN
					// Fehler eintragen, aber trotzdem weiter machen
					Step.eErrorStep := Step.eStepNr;
					Step.nSubscriptionIndex := -1;
					Step.nErrorId := fbUA_EventItemAdd.ErrorID;
					Step.eStepNr := eSTEP_RD_GET_NODE_HDL_LIST;
				END_IF
			END_IF

		eSTEP_RD_GET_NODE_HDL_LIST:
			// Die Handles für die ReadItems ermitteln
			brsmemset(ADR(fbUA_NodeGetHandleList), 0, SIZEOF(fbUA_NodeGetHandleList));
			fbUA_NodeGetHandleList.Execute := 1;
			fbUA_NodeGetHandleList.ConnectionHdl := nConnectionHandle;
			FOR nItemIndex:=0 TO nCLIENT_READ_ITEM_INDEX_MAX DO
				IF brsstrlen(ADR(ClientCfg.Read.Item[nItemIndex].NodeId.Identifier)) > 0 THEN
					brsmemcpy(ADR(fbUA_NodeGetHandleList.NodeIDs[nItemIndex]), ADR(ClientCfg.Read.Item[nItemIndex].NodeId), SIZEOF(UANodeID));
				ELSE
					EXIT;
				END_IF
			END_FOR
			fbUA_NodeGetHandleList.NodeIDCount := nItemIndex;
			fbUA_NodeGetHandleList.Timeout := tFB_TIMEOUT;
			Step.eStepNr := eSTEP_RD_GET_NODE_HDL_LIST_WAIT;

		eSTEP_RD_GET_NODE_HDL_LIST_WAIT:
			// Aufruf abwarten
			IF fbUA_NodeGetHandleList.Busy = 0 THEN
				fbUA_NodeGetHandleList.Execute := 0;
				IF fbUA_NodeGetHandleList.Done = 1 THEN
					// Daten speichern
					FOR nItemIndex := 0 TO nCLIENT_READ_ITEM_INDEX_MAX DO
						IF brsstrlen(ADR(ClientCfg.Read.Item[nItemIndex].NodeId.Identifier)) > 0 THEN
							fbUA_ReadList.NodeHdls[nItemIndex] := fbUA_NodeGetHandleList.NodeHdls[nItemIndex];
							fbUA_ReadList.NodeAddInfo[nItemIndex].AttributeId := UAAI_Value;
							brsstrcpy(ADR(asReadVars[nItemIndex]),  ADR(ClientCfg.Read.Item[nItemIndex].sVarName));
						ELSE
							EXIT;
						END_IF
					END_FOR
					fbUA_ReadList.NodeHdlCount := nItemIndex;
					Step.eStepNr := eSTEP_WR_GET_NODE_HDL_LIST;
				ELSIF fbUA_NodeGetHandleList.Error = 1 THEN
					// Fehler eintragen, aber trotzdem weiter machen
					Step.eErrorStep := Step.eStepNr;
					Step.nSubscriptionIndex := -1;
					IF fbUA_NodeGetHandleList.ErrorID <> 0 THEN
						Step.nItemIndex := -1;
						Step.nErrorId := fbUA_NodeGetHandleList.ErrorID;
					ELSE
						FOR nItemIndex :=0 TO MAX_INDEX_NODELIST DO
							IF fbUA_NodeGetHandleList.NodeErrorIDs[nItemIndex] <> 0 THEN
								Step.nItemIndex := nItemIndex;
								Step.nErrorId := fbUA_NodeGetHandleList.NodeErrorIDs[nItemIndex];
								EXIT;
							END_IF
						END_FOR
					END_IF
					nItemIndex := -1;
					Step.eStepNr := eSTEP_WR_GET_NODE_HDL_LIST;
				END_IF
			END_IF

		eSTEP_WR_GET_NODE_HDL_LIST:
			// Die Handles für die WriteItems ermitteln
			brsmemset(ADR(fbUA_NodeGetHandleList), 0, SIZEOF(fbUA_NodeGetHandleList));
			fbUA_NodeGetHandleList.Execute := 1;
			fbUA_NodeGetHandleList.ConnectionHdl := nConnectionHandle;
			FOR nItemIndex:=0 TO nCLIENT_WRITE_ITEM_INDEX_MAX DO
				IF brsstrlen(ADR(ClientCfg.Write.Item[nItemIndex].NodeId.Identifier)) > 0 THEN
					brsmemcpy(ADR(fbUA_NodeGetHandleList.NodeIDs[nItemIndex]), ADR(ClientCfg.Write.Item[nItemIndex].NodeId), SIZEOF(UANodeID));
				ELSE
					EXIT;
				END_IF
			END_FOR
			fbUA_NodeGetHandleList.NodeIDCount := nItemIndex;
			fbUA_NodeGetHandleList.Timeout := tFB_TIMEOUT;
			Step.eStepNr := eSTEP_WR_GET_NODE_HDL_LIST_WAIT;

		eSTEP_WR_GET_NODE_HDL_LIST_WAIT:
			// Aufruf abwarten
			IF fbUA_NodeGetHandleList.Busy = 0 THEN
				fbUA_NodeGetHandleList.Execute := 0;
				IF fbUA_NodeGetHandleList.Done = 1 THEN
					// Daten speichern
					FOR nItemIndex := 0 TO nCLIENT_WRITE_ITEM_INDEX_MAX DO
						IF brsstrlen(ADR(ClientCfg.Write.Item[nItemIndex].NodeId.Identifier)) > 0 THEN
							fbUA_WriteList.NodeHdls[nItemIndex] := fbUA_NodeGetHandleList.NodeHdls[nItemIndex];
							fbUA_WriteList.NodeAddInfo[nItemIndex].AttributeId := UAAI_Value;
							brsstrcpy(ADR(asWriteVars[nItemIndex]),  ADR(ClientCfg.Write.Item[nItemIndex].sVarName));
						ELSE
							EXIT;
						END_IF
					END_FOR
					fbUA_WriteList.NodeHdlCount := nItemIndex;
					Step.eStepNr := eSTEP_METH_GET_HANDLES;
				ELSIF fbUA_NodeGetHandleList.Error = 1 THEN
					// Fehler eintragen, aber trotzdem weiter machen
					Step.eErrorStep := Step.eStepNr;
					Step.nSubscriptionIndex := -1;
					IF fbUA_NodeGetHandleList.ErrorID <> 0 THEN
						Step.nItemIndex := -1;
						Step.nErrorId := fbUA_NodeGetHandleList.ErrorID;
					ELSE
						FOR nItemIndex :=0 TO MAX_INDEX_NODELIST DO
							IF fbUA_NodeGetHandleList.NodeErrorIDs[nItemIndex] <> 0 THEN
								Step.nItemIndex := nItemIndex;
								Step.nErrorId := fbUA_NodeGetHandleList.NodeErrorIDs[nItemIndex];
								EXIT;
							END_IF
						END_FOR
					END_IF
					nItemIndex := -1;
					Step.eStepNr := eSTEP_METH_GET_HANDLES;
				END_IF
			END_IF

		eSTEP_METH_GET_HANDLES:
			nMethodIndex := -1; // Mit der ersten Method beginnen
			Step.eStepNr := eSTEP_METH_GET_HANDLE;

		eSTEP_METH_GET_HANDLE:
			// Nächstes Method-Handle ermitteln
			nMethodIndex := nMethodIndex + 1;
			IF nMethodIndex <= nCLIENT_METHODS_INDEX_MAX THEN
				brsmemset(ADR(fbUA_MethodGetHandle), 0, SIZEOF(fbUA_MethodGetHandle));
				fbUA_MethodGetHandle.Execute := 1;
				fbUA_MethodGetHandle.ConnectionHdl := nConnectionHandle;
				brsmemcpy(ADR(fbUA_MethodGetHandle.ObjectNodeID), ADR(ClientCfg.Methods.Method[nMethodIndex].ObjectNodeId), SIZEOF(UANodeID));
				brsmemcpy(ADR(fbUA_MethodGetHandle.MethodNodeID), ADR(ClientCfg.Methods.Method[nMethodIndex].MethodNodeId), SIZEOF(UANodeID));
				fbUA_MethodGetHandle.Timeout := tFB_TIMEOUT;
				Step.eStepNr := eSTEP_METH_GET_HANDLE_WAIT;
			ELSE
				// Alle Method-Handles ermittelt
				IF Step.nErrorId <> 0 THEN
					Step.eStepNr := eSTEP_PAR_ERROR;
				ELSE
					Step.eStepNr := eSTEP_RUNNING;
				END_IF
			END_IF

		eSTEP_METH_GET_HANDLE_WAIT:
			// Aufruf abwarten
			IF fbUA_MethodGetHandle.Busy = 0 THEN
				fbUA_MethodGetHandle.Execute := 0;
				IF fbUA_MethodGetHandle.Done = 1 THEN
					anMethodHandles[nMethodIndex] := fbUA_MethodGetHandle.MethodHdl;
					Step.eStepNr := eSTEP_METH_GET_HANDLE;
				ELSIF fbUA_MethodGetHandle.Error = 1 THEN
					// Fehler eintragen, aber trotzdem weiter machen
					Step.eErrorStep := Step.eStepNr;
					Step.nSubscriptionIndex := -1;
					Step.nItemIndex := nMethodIndex;
					Step.nErrorId := fbUA_MethodGetHandle.ErrorID;
					Step.eStepNr := eSTEP_METH_GET_HANDLE;
				END_IF
			END_IF

		// -----------------------------------------------------------------------------------------------------------------------------------------------
		eSTEP_RUNNING:
			IF fbUA_ConnectionGetStatus.Execute = 1 THEN
				IF ConnectionStatus.eConnectionStatus <> UACS_Connected THEN
					// Der Server ist nicht mehr verbunden. In diesem Fall kann die Verbindung später vom Client automatisch wieder komplett reastauriert, wenn der Server wieder erreichbar ist.
					Step.eStepNr := eSTEP_CONNECTION_ERROR;
				ELSE
					// Trigger für zyklisches Lesen + Schreiben
					fbTrigger.IN := 1;
					IF fbTrigger.Q = 1 THEN
						fbTrigger.IN := 0;
						Step.eStepNr := eSTEP_READ_LIST;
					END_IF
				END_IF
			END_IF

		eSTEP_PAR_ERROR:
		// Es liegt eine Parameter-Fehler vor, bei dem die Schrittkette nicht weiter abgearbeitet werden kann.
		// Der falsche Parameter muss behoben werden.
		// Dieser ist unter der Struktur 'Step' einsehbar und kann in der AS-Hilfe nachgeschlagen werden.
		// Tipp: Die ErrorId sollte in Hexadezimal-Format angezeigt werden, da die OpcUa-Fehler immer als Hex dokumentiert werden.

		eSTEP_CONNECTION_ERROR:
			IF fbUA_ConnectionGetStatus.Execute = 1 THEN
				IF ConnectionStatus.eConnectionStatus = UACS_Connected THEN
					// Die Verbindung konnte vom Client automatisch wieder komplett reastauriert werden (mit allen Subscriptions und MonitoredItems)
					Step.eStepNr := eSTEP_RUNNING;
				END_IF
			END_IF

		// -----------------------------------------------------------------------------------------------------------------------------------------------
		eSTEP_READ_LIST:
			// Achtung: Zyklisches Lesen (Polling) sollte niemals in einer Applikation implementiert werden! Stattdessen sollte unbedingt Subscription verwendet werden.
			// Dieses Beispiel soll lediglich die Besetzung des FB's veranschaulichen.
			IF ConnectionStatus.eConnectionStatus <> UACS_Connected THEN
				Step.eStepNr := eSTEP_RUNNING;
			ELSE
				fbUA_ReadList.Execute := 1;
				fbUA_ReadList.ConnectionHdl := nConnectionHandle;
				fbUA_ReadList.Timeout := tFB_TIMEOUT;
				// Unter ST können IN/OUT-Elemente nicht direkt angegeben werden, sondern nur beim FB-Aufruf (siehe unten)
				// Der Eingang 'Variables' wird deshalb beim Aufruf übergeben
				Step.eStepNr := eSTEP_READ_LIST_WAIT;
			END_IF

		eSTEP_READ_LIST_WAIT:
			// Aufruf abwarten
			IF ConnectionStatus.eConnectionStatus <> UACS_Connected THEN
				fbUA_ReadList.Execute := 0;
				Step.eStepNr := eSTEP_RUNNING;
			ELSE
				IF fbUA_ReadList.Busy = 0 THEN
					fbUA_ReadList.Execute := 0;
					IF fbUA_ReadList.Error = 1 THEN
						// Fehler eintragen, aber trotzdem weiter machen
						Step.eErrorStep := Step.eStepNr;
						Step.nSubscriptionIndex := -1;
						IF fbUA_ReadList.ErrorID <> 0 THEN
							Step.nItemIndex := -1;
							Step.nErrorId := fbUA_ReadList.ErrorID;
						ELSE
							FOR nItemIndex := 0 TO nCLIENT_READ_ITEM_INDEX_MAX DO
								IF fbUA_ReadList.NodeErrorIDs[nItemIndex] <> 0 THEN
									Step.nItemIndex := nItemIndex;
									Step.nErrorId := fbUA_ReadList.NodeErrorIDs[nItemIndex];
									EXIT;
								END_IF
							END_FOR
						END_IF
					END_IF
					Step.eStepNr := eSTEP_WRITE_LIST;
				END_IF
			END_IF

		eSTEP_WRITE_LIST:
			IF ConnectionStatus.eConnectionStatus <> UACS_Connected THEN
				Step.eStepNr := eSTEP_RUNNING;
			ELSE
				fbUA_WriteList.Execute := 1;
				fbUA_WriteList.ConnectionHdl := nConnectionHandle;
				fbUA_WriteList.Timeout := tFB_TIMEOUT;
				// Unter ST können IN/OUT-Elemente nicht direkt angegeben werden, sondern nur beim FB-Aufruf (siehe unten)
				// Der Eingang 'Variables' wird deshalb beim Aufruf übergeben
				Step.eStepNr := eSTEP_WRITE_LIST_WAIT;
			END_IF

		eSTEP_WRITE_LIST_WAIT:
			// Aufruf abwarten
			IF ConnectionStatus.eConnectionStatus <> UACS_Connected THEN
				fbUA_WriteList.Execute := 0;
				Step.eStepNr := eSTEP_RUNNING;
			ELSE
				IF fbUA_WriteList.Busy = 0 THEN
					fbUA_WriteList.Execute := 0;
					IF fbUA_WriteList.Error = 1 THEN
						// Fehler eintragen, aber trotzdem weiter machen
						Step.eErrorStep := Step.eStepNr;
						Step.nSubscriptionIndex := -1;
						IF fbUA_WriteList.ErrorID <> 0 THEN
							Step.nItemIndex := -1;
							Step.nErrorId := fbUA_WriteList.ErrorID;
						ELSE
							FOR nItemIndex := 0 TO nCLIENT_WRITE_ITEM_INDEX_MAX DO
								IF fbUA_WriteList.NodeErrorIDs[nItemIndex] <> 0 THEN
									Step.nItemIndex := nItemIndex;
									Step.nErrorId := fbUA_WriteList.NodeErrorIDs[nItemIndex];
									EXIT;
								END_IF
							END_FOR
						END_IF
					END_IF
					Step.eStepNr := eSTEP_CALL_METH_CALC;
				END_IF
			END_IF

		eSTEP_CALL_METH_CALC:
			// Aufruf der Methode 'Calculate'
			IF ConnectionStatus.eConnectionStatus <> UACS_Connected THEN
				Step.eStepNr := eSTEP_RUNNING;
			ELSE
				fbUA_MethodCall.Execute := 1;
				fbUA_MethodCall.ConnectionHdl := nConnectionHandle;
				fbUA_MethodCall.MethodHdl := anMethodHandles[0];
				fbUA_MethodCall.Timeout := tFB_TIMEOUT;
				// Unter ST können IN/OUT-Elemente nicht direkt angegeben werden, sondern nur beim FB-Aufruf (siehe unten)
				// Eingänge mit Zufallszahlen besetzen
				MethCalculateArgs.In.nVal0 := BrbGetRandomDint(1, 10);
				MethCalculateArgs.In.nVal1 := BrbGetRandomDint(1, 10);
				FOR nItemIndex :=0 TO nMETHOD_CALC_ARRAY_INDEX_MAX DO
					MethCalculateArgs.In.anArray[nItemIndex] := DINT_TO_INT(BrbGetRandomDint(1, 10));
				END_FOR
				Step.eStepNr := eSTEP_CALL_METH_CALC_WAIT;
			END_IF

		eSTEP_CALL_METH_CALC_WAIT:
			// Aufruf abwarten
			IF ConnectionStatus.eConnectionStatus <> UACS_Connected THEN
				fbUA_MethodCall.Execute := 0;
				Step.eStepNr := eSTEP_RUNNING;
			ELSE
				IF fbUA_MethodCall.Busy = 0 THEN
					fbUA_MethodCall.Execute := 0;
					IF fbUA_MethodCall.Done = 1 THEN
						// Hier könnten die Ausgangs-Argumente ausgewertet werden
					ELSIF fbUA_MethodCall.Error = 1 THEN
						// Fehler eintragen, aber trotzdem weiter machen
						Step.eErrorStep := Step.eStepNr;
						Step.nSubscriptionIndex := -1;
						Step.nItemIndex := 0;
						Step.nErrorId := fbUA_MethodCall.ErrorID;
					END_IF
					Step.eStepNr := eSTEP_RUNNING;
				END_IF
			END_IF

	END_CASE

	// Der Verbindungs-Status sollte zyklisch geprüft werden
	fbUA_ConnectionGetStatus.Execute := (nConnectionHandle <> 0);
	fbUA_ConnectionGetStatus.ConnectionHdl := nConnectionHandle;
	fbUA_ConnectionGetStatus.Timeout := tFB_TIMEOUT;
	fbUA_ConnectionGetStatus();
	IF fbUA_ConnectionGetStatus.Done = 1 THEN
		ConnectionStatus.eConnectionStatus := fbUA_ConnectionGetStatus.ConnectionStatus;
		ConnectionStatus.eServerState := fbUA_ConnectionGetStatus.ServerState;
		ConnectionStatus.eServerLevel := fbUA_ConnectionGetStatus.ServiceLevel;
		fbUA_ConnectionGetStatus.Execute := 0;
		fbUA_ConnectionGetStatus();
	ELSIF fbUA_ConnectionGetStatus.Error = 1 THEN
		fbUA_ConnectionGetStatus.Execute := 0;
		fbUA_ConnectionGetStatus();
	END_IF
	IF nConnectionHandle = 0 THEN
		ConnectionStatus.eConnectionStatus := UACS_Shutdown;
		ConnectionStatus.eServerState := UASS_Unknown;
		ConnectionStatus.eServerLevel := 0;
	END_IF

	// Bearbeitung des EventItems (muss gemacht werden, um Events zu empfangen)
	fbUA_EventItemOperate.Execute := (fbUA_EventItemAdd.SubscriptionHdl <> 0 AND fbUA_EventItemAdd.EventItemHdl <> 0);
	fbUA_EventItemOperate.SubscriptionHdl := fbUA_EventItemAdd.SubscriptionHdl;
	fbUA_EventItemOperate.EventItemHdl := fbUA_EventItemAdd.EventItemHdl;
	fbUA_EventItemOperate.Timeout := tFB_TIMEOUT;
	fbUA_EventItemOperate();
	IF fbUA_EventItemOperate.Busy = 0 THEN
		IF fbUA_EventItemOperate.Done = 1 THEN
			IF fbUA_EventItemOperate.EventProcessed = 1 THEN
				// Es wurde ein Event empfangen
				ReceivedEvent.nReceivedCount := ReceivedEvent.nReceivedCount + 1;
				// Das Feld EventId wird in einen Hex-String gewandelt
				BrbUsintArrayToHex(ADR(ReceivedEvent.EventId.Data), ReceivedEvent.EventId.Length, ReceivedEvent.sEventIdHex, SIZEOF(ReceivedEvent.sEventIdHex), 0);
			END_IF
		ELSIF fbUA_EventItemOperate.Error = 1 THEN
			// In diesem Beispiel gibt es keine Fehlerbehandlung
		END_IF
		// Baustein für einen erneuten Aufruf zurücksetzen
		fbUA_EventItemOperate.Execute := 0;
		fbUA_EventItemOperate();
	END_IF

	// Aufruf aller sonstigen PlcOpen-Funktionsblöcke
	fbUA_Connect();
	fbUA_GetNamespaceIndex();
	fbUA_SubscriptionCreate(PublishingInterval := tSubscriptionPublishingInterval);
	fbUA_NodeGetHandleList();
	fbUA_MonitoredItemAddList(Variables := asMonitoredItemVarNames, MonitoringSettings := aMonitoredItemParameter, ValuesChanged := abMonItemValuesChanged, RemainingValueCount := anMonItemRemainingValueCount, TimeStamps := adtMonItemTimeStamps, NodeQualityIDs := anMonItemNodeQualityId);
	fbUA_NodeGetHandle();
	fbUA_EventItemAdd(EventFields := ClientCfg.Subscriptions.SubEvt.EventFieldVarNames);
	fbUA_MethodGetHandle();
	fbTrigger();
	fbUA_ReadList(Variables := asReadVars);
	fbUA_WriteList(Variables := asReadVars);
	fbUA_MethodCall(InputArguments := ClientCfg.Methods.Method[0].ArgumentsIn, OutputArguments := ClientCfg.Methods.Method[0].ArgumentsOut);

END_PROGRAM

PROGRAM _EXIT
	// Beim Überladen des Tasks wird zuerst der EXIT des alten Tasks ausgeführt und dieser dann gelöscht. Erst dann
	// wird der neue Task ausgeführt.
	// Solange die SPS nicht neu gestartet wird, wäre die Verbindung des alten Tasks immer noch vorhanden. Deshalb
	// sollte sie hier beeendet werden. Dabei werden alle angelegte Ressourcen (Verbindung, Subscriptions, MonitoredItems) sowohl beim Client als
	// auch beim Server aus dem Speicher gelöscht.
	// Auftretende Fehler müssen nicht ausgewertet werden. Deshalb wird nur auf Busy=0 gewartet.
	IF nConnectionHandle <> 0 THEN
		fbUA_Disconnect.Execute := 1;
		fbUA_Disconnect.ConnectionHdl := nConnectionHandle;
		fbUA_Disconnect.Timeout := tFB_TIMEOUT;
		REPEAT
			fbUA_Disconnect();
		UNTIL
			fbUA_Disconnect.Busy = 0
		END_REPEAT;
	END_IF
END_PROGRAM
```

#### ClientST.var - Local variables
```iecst
VAR
	bStartClient : BOOL;
	Step : Step_TYP;
	ClientCfg : ClientCfgTYP;
	fbUA_ConnectionGetStatus : UA_ConnectionGetStatus;
	ConnectionStatus : ClientConnectionStatus_TYP;
	fbUA_Connect : UA_Connect;
	nConnectionHandle : DWORD;
	fbUA_Disconnect : UA_Disconnect;
	fbUA_GetNamespaceIndex : UA_GetNamespaceIndex;
	fbUA_SubscriptionCreate : UA_SubscriptionCreate;
	nSubscriptionIndex : INT;
	tSubscriptionPublishingInterval : TIME;
	fbUA_NodeGetHandleList : UA_NodeGetHandleList;
	fbUA_MonitoredItemAddList : UA_MonitoredItemAddList;
	nItemIndex : INT;
	asMonitoredItemVarNames : ARRAY[0..MAX_INDEX_MONITORLIST] OF STRING[nVAR_NAME_CHAR_MAX];
	MonitoredItemParameter : UAMonitoringParameters;
	aMonitoredItemParameter : ARRAY[0..MAX_INDEX_MONITORLIST] OF UAMonitoringParameters;
	abMonItemValuesChanged : ARRAY[0..MAX_INDEX_MONITORLIST] OF BOOL;
	anMonItemRemainingValueCount : ARRAY[0..MAX_INDEX_MONITORLIST] OF UINT;
	adtMonItemTimeStamps : ARRAY[0..MAX_INDEX_MONITORLIST] OF DATE_AND_TIME;
	anMonItemNodeQualityId : ARRAY[0..MAX_INDEX_MONITORLIST] OF DWORD;
	ClientVarsSubscription : OpcUaTestDatatypes_TYP;
	fbUA_NodeGetHandle : UA_NodeGetHandle;
	fbUA_EventItemAdd : UA_EventItemAdd;
	fbTrigger : TON;
	fbUA_ReadList : UA_ReadList;
	asReadVars : ARRAY[0..MAX_INDEX_NODELIST] OF STRING[nVAR_NAME_CHAR_MAX];
	fbUA_WriteList : UA_WriteList;
	asWriteVars : ARRAY[0..MAX_INDEX_NODELIST] OF STRING[nVAR_NAME_CHAR_MAX];
	ClientVarsRead : OpcUaTestDatatypes_TYP;
	fbUA_MethodGetHandle : UA_MethodGetHandle;
	anMethodHandles : ARRAY[0..nCLIENT_METHODS_INDEX_MAX] OF DWORD;
	nMethodIndex : INT;
	fbUA_MethodCall : UA_MethodCall;
	MethCalculateArgs : MethCalculateArgs_TYP;
	fbUA_EventItemOperate : UA_EventItemOperate;
	ReceivedEvent : ProgressEvent_TYP;
END_VAR
```

### Package Logical/Tasks/OpcUaAny - Variablen für OpcUaAny-Client

### ReadMe.txt
```
Der OpcUaAny-Client ist als HW-Modul an der Ethernet-Schnittstelle eingefügt.
Er repräsentiert einen Server als IO-Modul und wird auch als 'normales' IO-Modul parametriert. Bedient
wird er automatisch durch einen im Betriebssystem integrierten Client.

Allgemeine Konfiguration:
	Die Einstellung 'Module supervised' sollte auf 'off' stehen. Sie verhält sie genauso wie bei jedem anderen
	IO-Modul. Das bedeutet, wenn sie auf 'on' steht und das Modul (also der Server) nicht erreicht wird, geht
	die SPS in den ServiceMode!
	Durch die Einstellung 'Server Diagnostics' werden Diagnose-Werte zur Verfügung gestellt, welche auf
	Variablen gemappt werden können (siehe IO-Mapping).
	Bei den Security-Einstellungen ist die SSL-Config angegeben, welche auch schon für den Lib-Client verwendet
	wird (Zertifikat mit 50 Jahren Laufzeit). Auch hier gilt: Wenn kein Zertifikat angegeben wird, wird
	automatisch eines mit einer Laufzeit von 10 Jahren angelegt.
	Ausserdem ist hier der Benutzer eingestellt, mit dem sich der Client am Server anmeldet.

Kanal-Konfiguration:
	Es wurden für dieses Beispiel je 3 Eingangs- und 3 Ausgangs-Kanäle angelegt. Eingänge dienen dem Lesen vom
	Server (genauer gesagt Abonnieren als MonitoredItems in Subscription(s)), Ausgänge dienen dem zyklischen
	Schreiben auf den Server.

	Zum Angeben des Knotens wird dabei nicht wie im Lib-Client eine NodeId verwendet, sondern die Einstellung
	'Browse path', welche eine alternative Addressierung darstellt. Sie muss den korrekten Browse-Pfad des zu
	addressierenden Knotens enthalten.
	Er besteht aus einzelnen Elementen, welche durch '/' getrennt sind und jeweils einen Knoten der Hierarchie
	darstellen. Ein Element enthält den Wert des Attributs 'BrowseName' des Knotens. Dieser wiederum besteht aus dem
	Namespace-Index und dann durch Doppelpunkt getrennt dem Knotennamen. Um Sonderzeichen trotzdem auch im
	eigentlichen Namen verwenden zu können, werden diese innerhalb des Pfades mit einem '&' als Prefix gekennzeichnet.
	Folgende Sonderzeichen werden gekennzeichnet:
		Zeichen			Ersetzung
		&						&&
		!						&!
		#						&#
		:						&:
		>						&>
		<						&<
		.						&.
		/						&/

	Somit ergibt z.B. bei B&R folgender Browse-Pfad:
	/0:Root/0:Objects/4:PLC/4:Modules/7:&:&:/7:OpcUaAny/7:Data/7:Read/7:Server/7:nUsint
	|																	|				|						|
	|																	|				|						+---	Ab hier beginnt der Variablenname
	|																	|				+---------------	Hier steht der Taskname
	|																	+-----------------------	Die : des Namens werden mit Präfix '&' gekennzeichnet
	+---------------------------------------------------------	Dies ist der Beginn des hierarchischen Address-Baums
																															Er ist bei B&R immer gleich

	Bei Fremd-Herstellern anderer Server kann der Pfad anders lauten.
	Im Zweifelsfalle können die BrowseNames der einzelnen Knoten durch einen generischen Client wie z.B.
	'UAExpert' (frei im Internet erhältlicher Windows-UA-Client) herausgefunden werden.

IO-Mapping:
	Standard-Kanäle
		ModuleOk
			Verhält sich wie bei einem normalen IO-Modul: Wenn der Server nicht erreichbar ist oder die Verbindung
			abbricht, geht dieser Kanal auf 'False'. Sobald die Verbindung besteht, ist er 'True'.
		ConnectionLostCount, ClientErrorCount und LastClientError
			Immer vorhandene Diagnose-Datenpunkte. Wenn ein Parametrier-Fehler vorliegt (z.B. falscher Browse-Pfad), kann
			dies an 'LastClientError' gesehen werden.
		ServerViewCount, CurrentSessionCount usw.
			Nur dann vorhandene Diagnose-Datenpunkte, wenn die Einstellung 'Server Diagnostics' auf 'on' steht.

	Benutzerdefinierte Kanäle
		Hier können die Kanäle gemappt werden, welche in der Konfiguration parametriert wurden.

	Wichtig: Eine zu mappende Variable muss den zum Datenpunkt passenden Datentyp haben!

Variablen in diesem Beispiel
	Der Task 'OpcUaAny' ist in diesem Beispiel nur vorhanden, um Variablen bereit zu stellen, welche an die
	Datenpunkte gemappt werden können.

	Eingänge:
		Die Elemente der Struktur 'Data.Read.Server' werden im Task inkrementiert und vom Client abonniert. Die
		empfangenen Werte werden auf die Struktur 'Data.Read.Client' geschrieben.

	Ausgänge:
		Die Elemente der Struktur 'Data.Write.Client' werden im Task inkrementiert und vom Client geschrieben.
		Serverseitig addressiert sind dabei die Elemente der Struktur 'Data.Write.Server'.

Verbindungsabbruch
	Wie schon beim Lib-Client wird auch hier nach einem Verbindungsabbruch die gesamte Kommunikation wieder
	automatisch restauriert. Ob eine Verbindung besteht, kann über den Eingangs-Kanal 'ModuleOk' abgefragt werden.
```

### Program Logical/Tasks/OpcUaAny/OpcUaAny (ANSIC) - Variablen für OpcUaAny-Client

#### OpcUaAny.c - Implementation code
```c
#include <bur/plctypes.h>

#ifdef _DEFAULT_INCLUDES
	#include <AsDefault.h>
#endif

// NOLINTBEGIN(readability-*, bugprone-easily-swappable-parameters, bugprone-branch-clone, clang-diagnostic-invalid-utf8, clang-diagnostic-invalid-source-encoding, clang-diagnostic-pointer-arith, clang-diagnostic-strict-prototypes, clang-diagnostic-shadow, clang-diagnostic-bad-function-cast, clang-analyzer-security.insecureAPI.*, hicpp-uppercase-literal-suffix, hicpp-function-size, cppcoreguidelines-*, performance-*)

void _INIT Init(void)
{
	brsmemset((UDINT)&Data, 0, sizeof(Data));
}

void _CYCLIC Cyclic(void)
{
	// Ändern der Server-Daten, welche vom OpcUaAny-Client gelesen werden
	Data.Read.Server.nUsint += 1;
	Data.Read.Server.nUint += 1;
	Data.Read.Server.nUdint += 1;

	// Ändern der Client-Daten, welche auf den Server geschrieben werden
	Data.Write.Client.nUsint += 2;
	Data.Write.Client.nUint += 2;
	Data.Write.Client.nUdint += 2;
}

void _EXIT Exit(void)
{
}

// NOLINTEND(readability-*, bugprone-easily-swappable-parameters, bugprone-branch-clone, clang-diagnostic-invalid-utf8, clang-diagnostic-invalid-source-encoding, clang-diagnostic-pointer-arith, clang-diagnostic-strict-prototypes, clang-diagnostic-shadow, clang-diagnostic-bad-function-cast, clang-analyzer-security.insecureAPI.*, hicpp-uppercase-literal-suffix, hicpp-function-size, cppcoreguidelines-*, performance-*)
```

#### OpcUaAny.typ - Local data types
```iecst
TYPE
	DataVars_TYP : 	STRUCT
		nUsint : USINT;
		nUint : UINT;
		nUdint : UDINT;
	END_STRUCT;
	DataReadWrite_TYP : 	STRUCT
		Server : DataVars_TYP;
		Client : DataVars_TYP;
	END_STRUCT;
	Data_TYP : 	STRUCT
		Read : DataReadWrite_TYP;
		Write : DataReadWrite_TYP;
	END_STRUCT;
END_TYPE
```

#### OpcUaAny.var - Local variables
```iecst
VAR
	Data : Data_TYP;
END_VAR
```

### Package Logical/Tasks/BrbUa - Verwendung der Bibliothek BrbLibUa

### ReadMe.txt
```
Die kostenlose Bibliothek 'BrbLibUa' enthält nützliche Funktionen rund um das Thema OpcUa.
Sie ist in der enthaltenen Datei 'BrbLibUa - Dokumentation' komplett beschrieben.
Sie hat eine Abhängigkeit auf die Bibliothek 'BrbLib', welche allgemein nützliche Funktionen enthält.
Beide Bibliotheken können kostenlos genutzt werden, aber es besteht für den Anwender kein Anspruch auf Support, Wartung
oder Fehlerbehebung. Die Benutzung geschieht auf eigene Gefahr.

Viele der Funktionen sind hier beispielhaft verwendet und zeigen den Vorteil dieser Bibliothek im Gegensatz zur
herkömmlichen Programmierung. Dies bedeutet, dass viele der Funktionalitäten mit relativ wenig Aufwand implementiert
werden können.

Unter anderem wird hier mithilfe der Bibliothek ein OpcUa-Client implementiert, welcher dieselben Funktionalitäten hat
wie der herkömmlich programmierte Client in diesem Projekt (Task 'Clients').
Schon anhand des Vergleichs der Code-Längen der beiden Tasks kann die enorme Zeitersparnis erahnt werden, welche mit
der Bibliothek erreicht werden kann.
Zusätzlich ist das Abonnieren der Server-Info- und Server-Diagnose-Daten implementiert. Dies könnte auch herkömmlich gemacht
werden, da dazu nur die Abonnierung bestimmter Knoten nötig ist, welche komplexe Datentypen mit dynamischen Arrays haben.
Bequemerweise sind diese Datentypen in der Bibliothek schon vordefiniert. Deshalb und weil die Abonnierung hier keinen Code
benötigt, ist das Beispiel nur hier implementiert. Außerdem können interessante Informationen dazu in der Hilfe der Bibliothek
nachgelesen werden.

Auch server-seitig gibt es Unterstützung. So ist z.B. eine Methode mithilfe der Bibliothek implementiert, was ebenfalls
eine Ersparnis zur herkömmlichen Programmierung bringt.
Auch das Feuern von Events wird von der Bibliothek unterstützt.
```

### Package Logical/Tasks/BrbUa/BrbUaClient - Client-Implementierung mit BrbLibUa

### ReadMe.txt
```
Diese Client-Implementierung mithilfe der Bibliothek BrbLibUa enthält dieselbe Funktionalität wie der herkömmlich
programmierte Client in diesem Projekt (Task 'Clients').
Schon anhand des Vergleichs der Code-Längen der beiden Tasks kann die enorme Zeitersparnis erahnt werden, welche mit
der Bibliothek erreicht werden kann.

Hinweis: Als Beispiel zum Empfangen eines Events wurde das Event 'EventTransitionType' gewählt, welches auch von den
Tasks in 'BrbUaServer' gefeuert wird. Da es diesen Server-Task zweimal gibt (für ANSI-C und StructuredTest), wird dieses
Event von beiden Server-Tasks gefeuert und deshalb auch von beiden empfangen. Zum Test können die Client- bzw. Server-Tasks
der nicht benötigten Sprache deaktiviert werden.

Zusätzlich ist das Abonnieren der Server-Diagnose-Daten implementiert. Dies könnte auch herkömmlich gemacht werden, da
dazu nur die Abonnierung bestimmter Knoten nötig ist, welche komplexe Datentypen mit dynamischen Arrays haben. Bequemerweise
sind diese Datentypen in der Bibliothek schon vordefiniert. Deshalb und weil die Abonnierung hier keinen Code benötigt, ist
das Beispiel nur hier implementiert. Außerdem können interessante Informationen dazu in der Hilfe der Bibliothek nachgelesen
werden.
```

### Package Logical/Tasks/BrbUa/BrbUaClient/BrbUaCltC - Client-Implementierung mit BrbLibUa in ANSI-C

### Data object Logical/Tasks/BrbUa/BrbUaClient/BrbUaCltC/BrbCltDatC (Simple) - Konfiguration des BrbUa-Clients für ANSI_C

#### DataObject.dat
```
;Konfiguration des BrbUa-Clients für ANSI-C

;Connection (Endpoint-Url wird im Programm gesetzt, nicht angegebene Parameter bleiben auf Default-Werten)
"§CONNECTION: SessionName=BrbUaClientC, AppName=AppBrbUaClientC, CertStore=SslCfgOpcUaClient, UserToken=1, TokenPar1=Admin, TokenPar2=admin, Locales=de;en"

;Namespaces
"§NAMESPACE: Uri=http://opcfoundation.org/UA/"
"§NAMESPACE: Uri=http://opcfoundation.org/UA/DI/"
"§NAMESPACE: Uri=http://br-automation.com/OpcUa/PLC/"
"§NAMESPACE: Uri=http://br-automation.com/OpcUa/PLC/PV/"

;NodeHandles
"§NODEHANDLE: Ns=3, Id=::BrbUaSrvC:VarsLocal.ReadOnly.nUdint"
"§NODEHANDLE: Ns=3, Id=::BrbUaSrvC:VarsLocal.ReadOnly.nDint"
"§NODEHANDLE: Ns=3, Id=::BrbUaSrvC:VarsLocal.ReadOnly.anInt"
"§NODEHANDLE: Ns=3, Id=::BrbUaSrvC:VarsLocal.WriteOnly.nUdint"
"§NODEHANDLE: Ns=3, Id=::BrbUaSrvC:VarsLocal.WriteOnly.nDint"
"§NODEHANDLE: Ns=3, Id=::BrbUaSrvC:VarsLocal.WriteOnly.anInt"

;ReadBlock 0
"§READBLOCK:"
"§READITEM: Ns=3, Id=::BrbUaSrvC:VarsLocal.ReadOnly.nUdint,		Var=::BrbUaCltC:ClientVarsRead.nUdint,	AttId=13"
"§READITEM: Ns=3, Id=::BrbUaSrvC:VarsLocal.ReadOnly.nDint,		Var=::BrbUaCltC:ClientVarsRead.nDint"
"§READITEM: Ns=3, Id=::BrbUaSrvC:VarsLocal.ReadOnly.anInt,		Var=::BrbUaCltC:ClientVarsRead.anInt"

;WriteBlock 0
"§WRITEBLOCK:"
"§WRITEITEM: Ns=3, Id=::BrbUaSrvC:VarsLocal.WriteOnly.nUdint,	Var=::BrbUaCltC:ClientVarsRead.nUdint,	AttId=13"
"§WRITEITEM: Ns=3, Id=::BrbUaSrvC:VarsLocal.WriteOnly.nDint,	Var=::BrbUaCltC:ClientVarsRead.nDint"
"§WRITEITEM: Ns=3, Id=::BrbUaSrvC:VarsLocal.WriteOnly.anInt,	Var=::BrbUaCltC:ClientVarsRead.anInt"

;Method 0 (Calculate)
"§METHOD: Ns=3, ObjectId=::BrbUaSrvC, MethodId=::BrbUaSrvC:Calculate, Timeout=1000"
"§METHODARGIN: Name=nValue0, 					Var=::BrbUaCltC:ClientMethCalculateArgs.In.nVal0"
"§METHODARGIN: Name=nValue1, 					Var=::BrbUaCltC:ClientMethCalculateArgs.In.nVal1"
"§METHODARGIN: Name=anArrayIn, 				Var=::BrbUaCltC:ClientMethCalculateArgs.In.anArray"
"§METHODARGOUT: Name=nAddition, 			Var=::BrbUaCltC:ClientMethCalculateArgs.Out.nAddition"
"§METHODARGOUT: Name=nMultiplication,	Var=::BrbUaCltC:ClientMethCalculateArgs.Out.nMultiplication"
"§METHODARGOUT: Name=anArrayOut, 			Var=::BrbUaCltC:ClientMethCalculateArgs.Out.anArray"

;Subscription 0 (Vars)
"§SUBSCRIPTION: Ena=1, Prio=200, PubInt=500"
"§MONITEM: Ns=3, Id=::BrbUaSrvC:VarsLocal.ReadOnly.bBool,			Var=::BrbUaCltC:ClientVarsSubscription.bBool"
"§MONITEM: Ns=3, Id=::BrbUaSrvC:VarsLocal.ReadOnly.nUsint,		Var=::BrbUaCltC:ClientVarsSubscription.nUsint"
"§MONITEM: Ns=3, Id=::BrbUaSrvC:VarsLocal.ReadOnly.nUint,			Var=::BrbUaCltC:ClientVarsSubscription.nUint"
"§MONITEM: Ns=3, Id=::BrbUaSrvC:VarsLocal.ReadOnly.nUdint,		Var=::BrbUaCltC:ClientVarsSubscription.nUdint"

;Subscription 1 (Vars)
"§SUBSCRIPTION: Ena=1, Prio=100, PubInt=1000"
"§MONITEM: Ns=3, Id=::BrbUaSrvC:VarsLocal.ReadOnly.nSint,			Var=::BrbUaCltC:ClientVarsSubscription.nSint"
"§MONITEM: Ns=3, Id=::BrbUaSrvC:VarsLocal.ReadOnly.nInt,			Var=::BrbUaCltC:ClientVarsSubscription.nInt"
"§MONITEM: Ns=3, Id=::BrbUaSrvC:VarsLocal.ReadOnly.nDint,			Var=::BrbUaCltC:ClientVarsSubscription.nDint"
"§MONITEM: Ns=3, Id=::BrbUaSrvC:VarsLocal.ReadOnly.rReal,			Var=::BrbUaCltC:ClientVarsSubscription.rReal"

;Subscription 2 (Vars)
"§SUBSCRIPTION: Ena=1, Prio=50, PubInt=2000"
"§MONITEM: Ns=3, Id=::BrbUaSrvC:VarsLocal.ReadOnly.rLongReal,		Var=::BrbUaCltC:ClientVarsSubscription.rLongReal"
"§MONITEM: Ns=3, Id=::BrbUaSrvC:VarsLocal.ReadOnly.sString,			Var=::BrbUaCltC:ClientVarsSubscription.sString"
"§MONITEM: Ns=3, Id=::BrbUaSrvC:VarsLocal.ReadOnly.tTime,				Var=::BrbUaCltC:ClientVarsSubscription.tTime"
"§MONITEM: Ns=3, Id=::BrbUaSrvC:VarsLocal.ReadOnly.dtDateTime,	Var=::BrbUaCltC:ClientVarsSubscription.dtDateTime"

;Subscription 3 (Event)
"§SUBSCRIPTION: Ena=1, Prio=250, PubInt=100"
"§EVTITEM: EvtNs=0, EvtId=2253, TypeNs=0, TypeId=2311, Timeout=1000, CallOperate=1"
"§EVTFIELD: FieldNs=0, FieldPath=EventId,										Var=::BrbUaCltC:ClientReceivedEvent.EventId"
"§EVTFIELD: FieldNs=0, FieldPath=EventType,									Var=::BrbUaCltC:ClientReceivedEvent.EventType"
"§EVTFIELD: FieldNs=0, FieldPath=LocalTime,									Var=::BrbUaCltC:ClientReceivedEvent.LocalTime"
"§EVTFIELD: FieldNs=0, FieldPath=Message,										Var=::BrbUaCltC:ClientReceivedEvent.Message"
"§EVTFIELD: FieldNs=0, FieldPath=ReceiveTime,								Var=::BrbUaCltC:ClientReceivedEvent.ReceiveTime"
"§EVTFIELD: FieldNs=0, FieldPath=Severity,									Var=::BrbUaCltC:ClientReceivedEvent.nSeverity"
"§EVTFIELD: FieldNs=0, FieldPath=SourceName,								Var=::BrbUaCltC:ClientReceivedEvent.sSourceName"
"§EVTFIELD: FieldNs=0, FieldPath=SourceNode,								Var=::BrbUaCltC:ClientReceivedEvent.SourceNode"
"§EVTFIELD: FieldNs=0, FieldPath=FromState,									Var=::BrbUaCltC:ClientReceivedEvent.FromState"
"§EVTFIELD: FieldNs=0, FieldPath=FromState,		FieldPath=Id,	Var=::BrbUaCltC:ClientReceivedEvent.nFromStateId"
"§EVTFIELD: FieldNs=0, FieldPath=ToState,										Var=::BrbUaCltC:ClientReceivedEvent.ToState"
"§EVTFIELD: FieldNs=0, FieldPath=ToState,			FieldPath=Id,	Var=::BrbUaCltC:ClientReceivedEvent.nToStateId"
"§EVTFIELD: FieldNs=0, FieldPath=Transition,								Var=::BrbUaCltC:ClientReceivedEvent.Transition"
"§EVTFIELD: FieldNs=0, FieldPath=Transition,	FieldPath=Id,	Var=::BrbUaCltC:ClientReceivedEvent.nTransitionId"

;Subscription 4 (ServerDiag)
"§SUBSCRIPTION: Ena=1, Prio=250, PubInt=1000"
"§MONITEM: Ns=0, Id=2255,		Var=::BrbUaCltC:ServerNamespacesArray"
"§MONITEM: Ns=0, Id=2256,		Var=::BrbUaCltC:ServerStatus"
"§MONITEM: Ns=0, Id=2275,		Var=::BrbUaCltC:ServerDiagData"
"§MONITEM: Ns=0, Id=3707,		Var=::BrbUaCltC:SessionDiagnosticsArray"
"§MONITEM: Ns=0, Id=3708,		Var=::BrbUaCltC:SessionSecurityDiagnosticsArray"
"§MONITEM: Ns=0, Id=2290,		Var=::BrbUaCltC:SubscriptionDiagnosticsArray"
```

### Program Logical/Tasks/BrbUa/BrbUaClient/BrbUaCltC/BrbUaCltC (ANSIC) - Client-Implementierung mit BrbLibUa in ANSI-C

#### BrbUaCltC.c - Implementation code
```c
#include <bur/plctypes.h>

#ifdef _DEFAULT_INCLUDES
	#include <AsDefault.h>
#endif

// NOLINTBEGIN(readability-*, bugprone-easily-swappable-parameters, bugprone-branch-clone, clang-diagnostic-invalid-utf8, clang-diagnostic-invalid-source-encoding, clang-diagnostic-pointer-arith, clang-diagnostic-strict-prototypes, clang-diagnostic-shadow, clang-diagnostic-bad-function-cast, clang-analyzer-security.insecureAPI.*, hicpp-uppercase-literal-suffix, hicpp-function-size, cppcoreguidelines-*, performance-*)

void _INIT Init(void)
{
	// Initialisierung des RunClients
	brsmemset((UDINT)&fbBrbUaRunClientInit, 0, sizeof(fbBrbUaRunClientInit));
	brsmemset((UDINT)&fbBrbUaRunClientCyclic, 0, sizeof(fbBrbUaRunClientCyclic));
	brsmemset((UDINT)&fbBrbUaRunClientExit, 0, sizeof(fbBrbUaRunClientExit));
	brsmemset((UDINT)&RunClient, 0, sizeof(RunClient));

	// Aufruf zum Initialisieren des RunClients
	brsstrcpy((UDINT)&RunClient.Cfg.sCfgDataObjName, (UDINT)&"BrbCltDatC");
	do
	{
		fbBrbUaRunClientInit.pRunClient = &RunClient;
		BrbUaRunClientInit(&fbBrbUaRunClientInit);
	} while(fbBrbUaRunClientInit.nStatus == eBRB_ERR_BUSY);

	// Wenn Verbindungs-Parameter im Datenobjekt nicht angeben sind, müssen sie nach dem Aufruf von RunClientInit, aber noch vor dem Connect-Kommando vom Programm gesetzt werden
	brsstrcpy((UDINT)&RunClient.Cfg.sServerEndpointUrl, (UDINT)&"opc.tcp://127.0.0.1:4840"); // z.B. Endpoint-Url besetzen

	RunClient.eCmd = eBRB_RCCLTCMD_CONNECT; // Sofort verbinden

	// Initialisierung des ReadBlock 0
	brsmemset((UDINT)&fbTimerReadBlock0, 0, sizeof(fbTimerReadBlock0));
	brsmemset((UDINT)&fbBrbUaRcReadBlock0, 0, sizeof(fbBrbUaRcReadBlock0));
	brsmemset((UDINT)&ClientVarsRead, 0, sizeof(ClientVarsRead));

	// Initialisierung des WriteBlock 0
	brsmemset((UDINT)&fbTimerWriteBlock0, 0, sizeof(fbTimerWriteBlock0));
	brsmemset((UDINT)&fbBrbUaRcWriteBlock0, 0, sizeof(fbBrbUaRcWriteBlock0));
	// Als Quelle der zu schreibenden Werte wird die Struktur 'ClientVarsRead' verwendet

	// Initialisierung der Methode 0 (Calculate)
	brsmemset((UDINT)&fbTimerCallMethodCalculate, 0, sizeof(fbTimerCallMethodCalculate));
	brsmemset((UDINT)&fbBrbUaRcCallMethodCalculate, 0, sizeof(fbBrbUaRcCallMethodCalculate));
	brsmemset((UDINT)&ClientMethCalculateArgs, 0, sizeof(ClientMethCalculateArgs));

	// Initialisierung der Variablen, die von den Subscriptions befüllt werden
	brsmemset((UDINT)&ClientVarsSubscription, 0, sizeof(ClientVarsSubscription));
	brsmemset((UDINT)&ClientReceivedEvent, 0, sizeof(ClientReceivedEvent));
	brsmemset((UDINT)&ServerNamespacesArray, 0, sizeof(ServerNamespacesArray));
	brsmemset((UDINT)&ServerStatus, 0, sizeof(ServerStatus));
	brsmemset((UDINT)&ServerDiagData, 0, sizeof(ServerDiagData));
	brsmemset((UDINT)&SessionDiagnosticsArray, 0, sizeof(SessionDiagnosticsArray));
	brsmemset((UDINT)&SessionSecurityDiagnosticsArray, 0, sizeof(SessionSecurityDiagnosticsArray));
	brsmemset((UDINT)&SubscriptionDiagnosticsArray, 0, sizeof(SubscriptionDiagnosticsArray));

	// Initialisierung der RunClient-Monitors
	brsmemset((UDINT)&RcMonitor, 0, sizeof(RcMonitor));

}

void _CYCLIC Cyclic(void)
{
	// Zyklischer Aufruf des RunClients
	if(RunClient.State.eClientState >= eBRB_RCCLTSTATE_INIT_DONE && RunClient.State.eClientState <= eBRB_RCCLTSTATE_EXITING)
	{
		fbBrbUaRunClientCyclic.pRunClient = &RunClient;
		BrbUaRunClientCyclic(&fbBrbUaRunClientCyclic);
	}

	// ReadBlock 0 lesen
	fbTimerReadBlock0.IN = (RunClient.State.eClientState == eBRB_RCCLTSTATE_CONNECTED);
	fbTimerReadBlock0.PT = 1000;
	TON(&fbTimerReadBlock0);
	if(fbTimerReadBlock0.Q == 1)
	{
		fbBrbUaRcReadBlock0.pRunClient = &RunClient;
		fbBrbUaRcReadBlock0.nReadBlockIndex = 0;
		BrbUaRcReadBlock(&fbBrbUaRcReadBlock0);
		if(fbBrbUaRcReadBlock0.nStatus != eBRB_ERR_BUSY)
		{
			// Timer neu triggern
			fbTimerReadBlock0.IN = 0;
			TON(&fbTimerReadBlock0);
		}
	}

	// WriteBlock 0 schreiben
	fbTimerWriteBlock0.IN = (RunClient.State.eClientState == eBRB_RCCLTSTATE_CONNECTED);
	fbTimerWriteBlock0.PT = 1000;
	TON(&fbTimerWriteBlock0);
	if(fbTimerWriteBlock0.Q == 1)
	{
		fbBrbUaRcWriteBlock0.pRunClient = &RunClient;
		fbBrbUaRcWriteBlock0.nWriteBlockIndex = 0;
		BrbUaRcWriteBlock(&fbBrbUaRcWriteBlock0);
		if(fbBrbUaRcWriteBlock0.nStatus != eBRB_ERR_BUSY)
		{
			// Timer neu triggern
			fbTimerWriteBlock0.IN = 0;
			TON(&fbTimerWriteBlock0);
		}
	}

	// Method 0 aufrufen (Calculate)
	fbTimerCallMethodCalculate.IN = (RunClient.State.eClientState == eBRB_RCCLTSTATE_CONNECTED);
	fbTimerCallMethodCalculate.PT = 1000;
	TON(&fbTimerCallMethodCalculate);
	if(fbTimerCallMethodCalculate.Q == 1)
	{
		fbBrbUaRcCallMethodCalculate.pRunClient = &RunClient;
		fbBrbUaRcCallMethodCalculate.nMethodIndex = 0;
		BrbUaRcCallMethod(&fbBrbUaRcCallMethodCalculate);
		if(fbBrbUaRcCallMethodCalculate.bInit == 1)
		{
			// Pro Aufruf einmalig Eingänge mit Zufallszahlen besetzen
			ClientMethCalculateArgs.In.nVal0 = BrbGetRandomDint(1, 10);
			ClientMethCalculateArgs.In.nVal1 = BrbGetRandomDint(1, 10);
			UINT nItemIndex = 0;
			for(nItemIndex=0; nItemIndex<=nMETHOD_CALC_ARRAY_INDEX_MAX; nItemIndex++)
			{
				ClientMethCalculateArgs.In.anArray[nItemIndex] = (INT)BrbGetRandomDint(1, 10);
			}
		}
		if(fbBrbUaRcCallMethodCalculate.nStatus != eBRB_ERR_BUSY)
		{
			// Call zurückgemeldet -> Timer neu triggern
			fbTimerCallMethodCalculate.IN = 0;
			TON(&fbTimerCallMethodCalculate);
		}
	}

	// Erkennen einer Wert-Änderung von Subscripton0, MonitoredItem1 (=nUsint)
	ClientReceivedMonItem.bValueChanged = BrbUaRcGetMiValueChanged(&RunClient, 0, 1, 0);
	if(ClientReceivedMonItem.bValueChanged == 1)
	{
		// Wert-Änderung wurde empfangen
		// Beispielsweise Zähler erhöhen
		ClientReceivedMonItem.nReceivedCount++;
		// Flag zurücksetzen
		BrbUaRcGetMiValueChanged(&RunClient, 0, 1, 1);
	}

	// Prüfen, ob Event von Subscripton3, EventItem0 empfangen wurde
	if(BrbUaRcGetEventItemReceived(&RunClient, 3, 0) == 1)
	{
		// Event wurde empfangen
		ClientReceivedEvent.nReceivedCount = BrbUaRcGetEventItemReceiveCount(&RunClient, 3, 0);
		// Das Feld EventId wird in einen Hex-String gewandelt
		BrbUsintArrayToHex((USINT*)&ClientReceivedEvent.EventId.Data, ClientReceivedEvent.EventId.Length, (STRING*)&ClientReceivedEvent.sEventIdHex, sizeof(ClientReceivedEvent.sEventIdHex), 0);
		// Das Feld ReceiveTime wird in einen Text gewandelt. Dabei wird mithilfe des Felds LocalTime von Utc-Zeit in lokale Server-Zeit umgerechnet
		BrbUaGetSrvTimeText(&ClientReceivedEvent.ReceiveTime, ClientReceivedEvent.sReceiveTime, sizeof(ClientReceivedEvent.sReceiveTime), ClientReceivedEvent.LocalTime.TimeOffset, "yyyy:mm:dd hh:MM:ss::milms:mic.µs:nanns");
	}

	// RunClient-Monitor
	BrbUaRcMonitor(&RunClient, &RcMonitor);

}

void _EXIT Exit(void)
{
	// Aufruf zum Exit des RunClients
	do
	{
		fbBrbUaRunClientExit.pRunClient = &RunClient;
		BrbUaRunClientExit(&fbBrbUaRunClientExit);
	} while(fbBrbUaRunClientExit.nStatus == eBRB_ERR_BUSY);
}

// NOLINTEND(readability-*, bugprone-easily-swappable-parameters, bugprone-branch-clone, clang-diagnostic-invalid-utf8, clang-diagnostic-invalid-source-encoding, clang-diagnostic-pointer-arith, clang-diagnostic-strict-prototypes, clang-diagnostic-shadow, clang-diagnostic-bad-function-cast, clang-analyzer-security.insecureAPI.*, hicpp-uppercase-literal-suffix, hicpp-function-size, cppcoreguidelines-*, performance-*)
```

#### BrbUaCltC.var - Local variables
```iecst
(*Client*)
(*Insert your comment here.*)
VAR
	RunClient : BrbUaRunClient_TYP;
	fbBrbUaRunClientInit : BrbUaRunClientInit;
	fbBrbUaRunClientCyclic : BrbUaRunClientCyclic;
	fbBrbUaRunClientExit : BrbUaRunClientExit;
	fbTimerReadBlock0 : TON;
	fbBrbUaRcReadBlock0 : BrbUaRcReadBlock;
	fbTimerWriteBlock0 : TON;
	fbBrbUaRcWriteBlock0 : BrbUaRcWriteBlock;
	fbTimerCallMethodCalculate : TON;
	fbBrbUaRcCallMethodCalculate : BrbUaRcCallMethod;
END_VAR
(*Application Variables*)
VAR
	ClientVarsSubscription : OpcUaTestDatatypes_TYP;
	ClientVarsRead : OpcUaTestDatatypes_TYP;
	ClientMethCalculateArgs : MethCalculateArgs_TYP;
	ClientReceivedMonItem : ClientReceivedMonItem_TYP;
	ClientReceivedEvent : TransitionEvent_TYP;
	ServerNamespacesArray : BrbUaServerNamespacesArray_TYP;
	ServerStatus : BrbUaServerStatus_TYP;
	ServerDiagData : BrbUaServerDiagData_TYP;
	SessionDiagnosticsArray : BrbUaSessDiagArray_TYP;
	SessionSecurityDiagnosticsArray : BrbUaSessSecDiagArray_TYP;
	SubscriptionDiagnosticsArray : BrbUaSubscriptDiagArray_TYP;
END_VAR
(*Monitor*)
VAR
	RcMonitor : BrbUaRcMonitor_TYP;
END_VAR
```

### Package Logical/Tasks/BrbUa/BrbUaClient/BrbUaCltST - Client-Implementierung mit BrbLibUa in ST

### Data object Logical/Tasks/BrbUa/BrbUaClient/BrbUaCltST/BrbCltDatST (Simple) - Konfiguration des BrbUa-Clients für ST

#### DataObject.dat
```
;Konfiguration des BrbUa-Clients für ST

;Connection (Endpoint-Url wird im Programm gesetzt, nicht angegebene Parameter bleiben auf Default-Werten)
"§CONNECTION: SessionName=BrbUaClientST, AppName=AppBrbUaClientST, CertStore=SslCfgOpcUaClient, UserToken=1, TokenPar1=Admin, TokenPar2=admin, Locales=de;en"

;Namespaces
"§NAMESPACE: Uri=http://opcfoundation.org/UA/"
"§NAMESPACE: Uri=http://opcfoundation.org/UA/DI/"
"§NAMESPACE: Uri=http://br-automation.com/OpcUa/PLC/"
"§NAMESPACE: Uri=http://br-automation.com/OpcUa/PLC/PV/"

;NodeHandles
"§NODEHANDLE: Ns=3, Id=::BrbUaSrvST:VarsLocal.ReadOnly.nUdint"
"§NODEHANDLE: Ns=3, Id=::BrbUaSrvST:VarsLocal.ReadOnly.nDint"
"§NODEHANDLE: Ns=3, Id=::BrbUaSrvST:VarsLocal.ReadOnly.anInt"
"§NODEHANDLE: Ns=3, Id=::BrbUaSrvST:VarsLocal.WriteOnly.nUdint"
"§NODEHANDLE: Ns=3, Id=::BrbUaSrvST:VarsLocal.WriteOnly.nDint"
"§NODEHANDLE: Ns=3, Id=::BrbUaSrvST:VarsLocal.WriteOnly.anInt"

;ReadBlock 0
"§READBLOCK:"
"§READITEM: Ns=3, Id=::BrbUaSrvST:VarsLocal.ReadOnly.nUdint,		Var=::BrbUaCltST:ClientVarsRead.nUdint,	AttId=13"
"§READITEM: Ns=3, Id=::BrbUaSrvST:VarsLocal.ReadOnly.nDint,			Var=::BrbUaCltST:ClientVarsRead.nDint"
"§READITEM: Ns=3, Id=::BrbUaSrvST:VarsLocal.ReadOnly.anInt,			Var=::BrbUaCltST:ClientVarsRead.anInt"

;WriteBlock 0
"§WRITEBLOCK:"
"§WRITEITEM: Ns=3, Id=::BrbUaSrvST:VarsLocal.WriteOnly.nUdint,		Var=::BrbUaCltST:ClientVarsRead.nUdint,	AttId=13"
"§WRITEITEM: Ns=3, Id=::BrbUaSrvST:VarsLocal.WriteOnly.nDint,			Var=::BrbUaCltST:ClientVarsRead.nDint"
"§WRITEITEM: Ns=3, Id=::BrbUaSrvST:VarsLocal.WriteOnly.anInt,			Var=::BrbUaCltST:ClientVarsRead.anInt"

;Method 0 (Calculate)
"§METHOD: Ns=3, ObjectId=::BrbUaSrvST, MethodId=::BrbUaSrvST:Calculate, Timeout=1000"
"§METHODARGIN: Name=nValue0, Var=::BrbUaCltST:ClientMethCalculateArgs.In.nVal0"
"§METHODARGIN: Name=nValue1, Var=::BrbUaCltST:ClientMethCalculateArgs.In.nVal1"
"§METHODARGIN: Name=anArrayIn, Var=::BrbUaCltST:ClientMethCalculateArgs.In.anArray"
"§METHODARGOUT: Name=nAddition, Var=::BrbUaCltST:ClientMethCalculateArgs.Out.nAddition"
"§METHODARGOUT: Name=nMultiplication, Var=::BrbUaCltST:ClientMethCalculateArgs.Out.nMultiplication"
"§METHODARGOUT: Name=anArrayOut, Var=::BrbUaCltST:ClientMethCalculateArgs.Out.anArray"

;Subscription 0 (Vars)
"§SUBSCRIPTION: Ena=1, Prio=200, PubInt=500"
"§MONITEM: Ns=3, Id=::BrbUaSrvST:VarsLocal.ReadOnly.bBool,			Var=::BrbUaCltST:ClientVarsSubscription.bBool"
"§MONITEM: Ns=3, Id=::BrbUaSrvST:VarsLocal.ReadOnly.nUsint,			Var=::BrbUaCltST:ClientVarsSubscription.nUsint"
"§MONITEM: Ns=3, Id=::BrbUaSrvST:VarsLocal.ReadOnly.nUint,			Var=::BrbUaCltST:ClientVarsSubscription.nUint"
"§MONITEM: Ns=3, Id=::BrbUaSrvST:VarsLocal.ReadOnly.nUdint,			Var=::BrbUaCltST:ClientVarsSubscription.nUdint"

;Subscription 1 (Vars)
"§SUBSCRIPTION: Ena=1, Prio=100, PubInt=1000"
"§MONITEM: Ns=3, Id=::BrbUaSrvST:VarsLocal.ReadOnly.nSint,			Var=::BrbUaCltST:ClientVarsSubscription.nSint"
"§MONITEM: Ns=3, Id=::BrbUaSrvST:VarsLocal.ReadOnly.nInt,				Var=::BrbUaCltST:ClientVarsSubscription.nInt"
"§MONITEM: Ns=3, Id=::BrbUaSrvST:VarsLocal.ReadOnly.nDint,			Var=::BrbUaCltST:ClientVarsSubscription.nDint"
"§MONITEM: Ns=3, Id=::BrbUaSrvST:VarsLocal.ReadOnly.rReal,			Var=::BrbUaCltST:ClientVarsSubscription.rReal"

;Subscription 2 (Vars)
"§SUBSCRIPTION: Ena=1, Prio=50, PubInt=2000"
"§MONITEM: Ns=3, Id=::BrbUaSrvST:VarsLocal.ReadOnly.rLongReal,	Var=::BrbUaCltST:ClientVarsSubscription.rLongReal"
"§MONITEM: Ns=3, Id=::BrbUaSrvST:VarsLocal.ReadOnly.sString,		Var=::BrbUaCltST:ClientVarsSubscription.sString"
"§MONITEM: Ns=3, Id=::BrbUaSrvST:VarsLocal.ReadOnly.tTime,			Var=::BrbUaCltST:ClientVarsSubscription.tTime"
"§MONITEM: Ns=3, Id=::BrbUaSrvST:VarsLocal.ReadOnly.dtDateTime,	Var=::BrbUaCltST:ClientVarsSubscription.dtDateTime"

;Subscription 3 (Event)
"§SUBSCRIPTION: Ena=1, Prio=250, PubInt=100"
"§EVTITEM: EvtNs=0, EvtId=2253, TypeNs=0, TypeId=2311, Timeout=1000, CallOperate=1"
"§EVTFIELD: FieldNs=0, FieldPath=EventId,										Var=::BrbUaCltST:ClientReceivedEvent.EventId"
"§EVTFIELD: FieldNs=7, FieldPath=EventType,									Var=::BrbUaCltST:ClientReceivedEvent.EventType"
"§EVTFIELD: FieldNs=0, FieldPath=LocalTime,									Var=::BrbUaCltST:ClientReceivedEvent.LocalTime"
"§EVTFIELD: FieldNs=0, FieldPath=Message,										Var=::BrbUaCltST:ClientReceivedEvent.Message"
"§EVTFIELD: FieldNs=0, FieldPath=ReceiveTime,								Var=::BrbUaCltST:ClientReceivedEvent.ReceiveTime"
"§EVTFIELD: FieldNs=0, FieldPath=Severity,									Var=::BrbUaCltST:ClientReceivedEvent.nSeverity"
"§EVTFIELD: FieldNs=0, FieldPath=SourceName,								Var=::BrbUaCltST:ClientReceivedEvent.sSourceName"
"§EVTFIELD: FieldNs=0, FieldPath=SourceNode,								Var=::BrbUaCltST:ClientReceivedEvent.SourceNode"
"§EVTFIELD: FieldNs=0, FieldPath=FromState,									Var=::BrbUaCltST:ClientReceivedEvent.FromState"
"§EVTFIELD: FieldNs=0, FieldPath=FromState,		FieldPath=Id,	Var=::BrbUaCltST:ClientReceivedEvent.nFromStateId"
"§EVTFIELD: FieldNs=0, FieldPath=ToState,										Var=::BrbUaCltST:ClientReceivedEvent.ToState"
"§EVTFIELD: FieldNs=0, FieldPath=ToState,			FieldPath=Id,	Var=::BrbUaCltST:ClientReceivedEvent.nToStateId"
"§EVTFIELD: FieldNs=0, FieldPath=Transition,								Var=::BrbUaCltST:ClientReceivedEvent.Transition"
"§EVTFIELD: FieldNs=0, FieldPath=Transition,	FieldPath=Id,	Var=::BrbUaCltST:ClientReceivedEvent.nTransitionId"

;Subscription 4 (ServerDiag)
"§SUBSCRIPTION: Ena=1, Prio=250, PubInt=1000"
"§MONITEM: Ns=0, Id=2255,		Var=::BrbUaCltST:ServerNamespacesArray"
"§MONITEM: Ns=0, Id=2256,		Var=::BrbUaCltST:ServerStatus"
"§MONITEM: Ns=0, Id=2275,		Var=::BrbUaCltST:ServerDiagData"
"§MONITEM: Ns=0, Id=3707,		Var=::BrbUaCltST:SessionDiagnosticsArray"
"§MONITEM: Ns=0, Id=3708,		Var=::BrbUaCltST:SessionSecurityDiagnosticsArray"
"§MONITEM: Ns=0, Id=2290,		Var=::BrbUaCltST:SubscriptionDiagnosticsArray"
```

### Program Logical/Tasks/BrbUa/BrbUaClient/BrbUaCltST/BrbUaCltST (IEC) - Client-Implementierung mit BrbLibUa in ST

#### BrbUaCltST.st - Init, cyclic, exit code
```iecst
PROGRAM _INIT
	// Initialisierung des Clients
	brsmemset(ADR(fbBrbUaRunClientInit), 0, SIZEOF(fbBrbUaRunClientInit));
	brsmemset(ADR(fbBrbUaRunClientCyclic), 0, SIZEOF(fbBrbUaRunClientCyclic));
	brsmemset(ADR(fbBrbUaRunClientExit), 0, SIZEOF(fbBrbUaRunClientExit));
	brsmemset(ADR(RunClient), 0, SIZEOF(RunClient));

	// Aufruf zum Initialisieren des Clients
	RunClient.Cfg.sCfgDataObjName := 'BrbCltDatS';
	REPEAT
		fbBrbUaRunClientInit.pRunClient := ADR(RunClient);
		fbBrbUaRunClientInit();
		UNTIL fbBrbUaRunClientInit.nStatus <> eBRB_ERR_BUSY
	END_REPEAT

	// Wenn Verbindungs-Parameter im Datenobjekt nicht angeben sind, müssen sie nach dem Aufruf von RunClientInit, aber noch vor dem Connect-Kommando vom Programm gesetzt werden
	RunClient.Cfg.sServerEndpointUrl := 'opc.tcp://127.0.0.1:4840/'; // z.B. Endpoint-Url besetzen
	RunClient.eCmd := eBRB_RCCLTCMD_CONNECT; // Sofort verbinden

	// Initialisierung des ReadBlock 0
	brsmemset(ADR(fbTimerReadBlock0), 0, SIZEOF(fbTimerReadBlock0));
	brsmemset(ADR(fbBrbUaRcReadBlock0), 0, SIZEOF(fbBrbUaRcReadBlock0));
	brsmemset(ADR(ClientVarsRead), 0, SIZEOF(ClientVarsRead));

	// Initialisierung des WriteBlock 0
	brsmemset(ADR(fbTimerWriteBlock0), 0, SIZEOF(fbTimerWriteBlock0));
	brsmemset(ADR(fbBrbUaRcWriteBlock0), 0, SIZEOF(fbBrbUaRcWriteBlock0));
	// Als Quelle der zu schreibenden Werte wird die Struktur 'ClientVarsRead' verwendet

	// Initialisierung der Methode 0 (Calculate)
	brsmemset(ADR(fbTimerCallMethodCalculate), 0, SIZEOF(fbTimerCallMethodCalculate));
	brsmemset(ADR(fbBrbUaRcCallMethodCalculate), 0, SIZEOF(fbBrbUaRcCallMethodCalculate));
	brsmemset(ADR(ClientMethCalculateArgs), 0, SIZEOF(ClientMethCalculateArgs));

	// Initialisierung der Variablen, die von den Subscriptions befüllt werden
	brsmemset(ADR(ClientVarsSubscription), 0, SIZEOF(ClientVarsSubscription));
	brsmemset(ADR(ClientReceivedEvent), 0, SIZEOF(ClientReceivedEvent));
	brsmemset(ADR(ServerNamespacesArray), 0, SIZEOF(ServerNamespacesArray));
	brsmemset(ADR(ServerStatus), 0, SIZEOF(ServerStatus));
	brsmemset(ADR(ServerDiagData), 0, SIZEOF(ServerDiagData));
	brsmemset(ADR(SessionDiagnosticsArray), 0, SIZEOF(SessionDiagnosticsArray));
	brsmemset(ADR(SessionSecurityDiagnosticsArray), 0, SIZEOF(SessionSecurityDiagnosticsArray));
	brsmemset(ADR(SubscriptionDiagnosticsArray), 0, SIZEOF(SubscriptionDiagnosticsArray));

	// Initialisierung der Monitors
	brsmemset(ADR(RcMonitor), 0, SIZEOF(RcMonitor));

END_PROGRAM

PROGRAM _CYCLIC

	// Zyklischer Aufruf des Clients
	IF RunClient.State.eClientState >= eBRB_RCCLTSTATE_INIT_DONE AND RunClient.State.eClientState <= eBRB_RCCLTSTATE_EXITING THEN
		fbBrbUaRunClientCyclic.pRunClient := ADR(RunClient);
		fbBrbUaRunClientCyclic();
	END_IF

	// ReadBlock 0 lesen
	fbTimerReadBlock0.IN := (RunClient.State.eClientState = eBRB_RCCLTSTATE_CONNECTED);
	fbTimerReadBlock0.PT := T#1s;
	fbTimerReadBlock0();
	IF fbTimerReadBlock0.Q = 1 THEN
		fbBrbUaRcReadBlock0.pRunClient := ADR(RunClient);
		fbBrbUaRcReadBlock0.nReadBlockIndex := 0;
		fbBrbUaRcReadBlock0();
		IF fbBrbUaRcReadBlock0.nStatus <> eBRB_ERR_BUSY THEN
			// Timer neu triggern
			fbTimerReadBlock0.IN := 0;
			fbTimerReadBlock0();
		END_IF
	END_IF

	// WriteBlock 0 schreiben
	fbTimerWriteBlock0.IN := (RunClient.State.eClientState = eBRB_RCCLTSTATE_CONNECTED);
	fbTimerWriteBlock0.PT := T#1s;
	fbTimerWriteBlock0();
	IF fbTimerWriteBlock0.Q = 1 THEN
		fbBrbUaRcWriteBlock0.pRunClient := ADR(RunClient);
		fbBrbUaRcWriteBlock0.nWriteBlockIndex := 0;
		fbBrbUaRcWriteBlock0();
		IF fbBrbUaRcWriteBlock0.nStatus <> eBRB_ERR_BUSY THEN
			// Timer neu triggern
			fbTimerWriteBlock0.IN := 0;
			fbTimerWriteBlock0();
		END_IF
	END_IF

	// Method 0 aufrufen (Calculate)
	fbTimerCallMethodCalculate.IN := (RunClient.State.eClientState = eBRB_RCCLTSTATE_CONNECTED);
	fbTimerCallMethodCalculate.PT := T#1s;
	fbTimerCallMethodCalculate();
	IF fbTimerCallMethodCalculate.Q = 1 THEN
		fbBrbUaRcCallMethodCalculate.pRunClient := ADR(RunClient);
		fbBrbUaRcCallMethodCalculate.nMethodIndex := 0;
		fbBrbUaRcCallMethodCalculate();
		IF fbBrbUaRcCallMethodCalculate.bInit = 1 THEN
			// Pro Aufruf einmalig Eingänge mit Zufallszahlen besetzen
			ClientMethCalculateArgs.In.nVal0 := BrbGetRandomDint(1, 10);
			ClientMethCalculateArgs.In.nVal1 := BrbGetRandomDint(1, 10);
			FOR nItemIndex :=0 TO nMETHOD_CALC_ARRAY_INDEX_MAX DO
				ClientMethCalculateArgs.In.anArray[nItemIndex] := DINT_TO_INT(BrbGetRandomDint(1, 10));
			END_FOR
		END_IF
		IF fbBrbUaRcCallMethodCalculate.nStatus <> eBRB_ERR_BUSY THEN
			// Call zurückgemeldet -> Timer neu triggern
			fbTimerCallMethodCalculate.IN := 0;
			fbTimerCallMethodCalculate();
		END_IF
	END_IF

	// Erkennen einer Wert-Änderung von Subscripton0, MonitoredItem1 (=nUsint)
	ClientReceivedMonItem.bValueChanged := BrbUaRcGetMiValueChanged(RunClient, 0, 1, 0);
	IF ClientReceivedMonItem.bValueChanged = 1 THEN
		// Wert-Änderung wurde empfangen
		// Beispielsweise Zähler erhöhen
		ClientReceivedMonItem.nReceivedCount := ClientReceivedMonItem.nReceivedCount + 1;
		// Flag zurücksetzen
		BrbUaRcGetMiValueChanged(RunClient, 0, 1, 1);
	END_IF

	// Prüfen, ob Event von Subscripton3, EventItem0 empfangen wurde
	IF BrbUaRcGetEventItemReceived(RunClient, 3, 0) = 1 THEN
		// Event wurde empfangen
		ClientReceivedEvent.nReceivedCount := BrbUaRcGetEventItemReceiveCount(RunClient, 3, 0);
		// Das Feld EventId wird in einen Hex-String gewandelt
		BrbUsintArrayToHex(ADR(ClientReceivedEvent.EventId.Data), ClientReceivedEvent.EventId.Length, ClientReceivedEvent.sEventIdHex, SIZEOF(ClientReceivedEvent.sEventIdHex), 0);
		// Das Feld ReceiveTime wird in einen Text gewandelt. Dabei wird mithilfe des Felds LocalTime von Utc-Zeit in lokale Server-Zeit umgerechnet
		BrbUaGetSrvTimeText(ClientReceivedEvent.ReceiveTime, ClientReceivedEvent.sReceiveTime, SIZEOF(ClientReceivedEvent.sReceiveTime), ClientReceivedEvent.LocalTime.TimeOffset, 'yyyy:mm:dd hh:MM:ss::milms:mic.µs:nanns');

	END_IF

	// RunClient-Monitor
	BrbUaRcMonitor(RunClient, RcMonitor);

END_PROGRAM

PROGRAM _EXIT
	// Aufruf zum Exit des RunClients
	REPEAT
		fbBrbUaRunClientExit.pRunClient := ADR(RunClient);
		fbBrbUaRunClientExit();
		UNTIL fbBrbUaRunClientExit.nStatus <> eBRB_ERR_BUSY
	END_REPEAT
END_PROGRAM
```

#### BrbUaCltST.var - Local variables
```iecst
(*Client*)
VAR
	RunClient : BrbUaRunClient_TYP;
	fbBrbUaRunClientInit : BrbUaRunClientInit;
	fbBrbUaRunClientCyclic : BrbUaRunClientCyclic;
	fbBrbUaRunClientExit : BrbUaRunClientExit;
	fbTimerReadBlock0 : TON;
	fbBrbUaRcReadBlock0 : BrbUaRcReadBlock;
	fbTimerWriteBlock0 : TON;
	fbBrbUaRcWriteBlock0 : BrbUaRcWriteBlock;
	fbTimerCallMethodCalculate : TON;
	fbBrbUaRcCallMethodCalculate : BrbUaRcCallMethod;
END_VAR
(*Application Variables*)
VAR
	nItemIndex : UINT;
	ClientVarsSubscription : OpcUaTestDatatypes_TYP;
	ClientVarsRead : OpcUaTestDatatypes_TYP;
	ClientMethCalculateArgs : MethCalculateArgs_TYP;
	ClientReceivedMonItem : ClientReceivedMonItem_TYP;
	ClientReceivedEvent : TransitionEvent_TYP;
	ServerNamespacesArray : BrbUaServerNamespacesArray_TYP;
	ServerStatus : BrbUaServerStatus_TYP;
	ServerDiagData : BrbUaServerDiagData_TYP;
	SessionDiagnosticsArray : BrbUaSessDiagArray_TYP;
	SessionSecurityDiagnosticsArray : BrbUaSessSecDiagArray_TYP;
	SubscriptionDiagnosticsArray : BrbUaSubscriptDiagArray_TYP;
END_VAR
(*Monitor*)
VAR
	RcMonitor : BrbUaRcMonitor_TYP;
END_VAR
```

### Package Logical/Tasks/BrbUa/BrbUaServer - Server-Implementierung mit BrbLibUa

### ReadMe.txt
```
Hier werden dieselben lokalen Variablen 'VarsLocal' zur Verfügung gestellt wie im Task 'ServerData'.
Auf sie wird im Task 'BrbUaClient' zugegriffen.
Zusätzlich wird der Umgang mit dem Datentyp "UAByteStringBrbEventId_TYP" gezeigt, welcher eine 16 Byte lange
EventId aufnimmt und veröffentlicht.

Ausserdem ist dieselbe Methode 'Calculate' implementiert wie im Task 'ServerMethods'.
Beachtenswert ist die Kürze des Codes. Statt einer kompletten Schrittkette kann die Methode in einem relativ
kleinen If-Then-Else-Block abgehandelt werden.

Auch das Feuern eines Events mithilfe des RunServers ist hier implementiert. Im Gegegsatz zur herkömmlichen
Programmierung (Tasks 'ServerEvents') wird hier aber nicht das Event 'ProgessType', sondern 'TransitionType'
gefeuert. Auch hier ist die Kürze des Codes ausschlaggebend.
```

### Package Logical/Tasks/BrbUa/BrbUaServer/BrbUaSrvC - Server-Implementierung mit BrbLibUa in ANSI-C

### Data object Logical/Tasks/BrbUa/BrbUaServer/BrbUaSrvC/BrbSrvDatC (Simple) - Konfiguration des BrbUa-Servers für ANSI_C

#### DataObject.dat
```
;Konfiguration des BrbUa-Servers für ANSI-C

;Namespaces
"§NAMESPACE: Uri=http://opcfoundation.org/UA/"
"§NAMESPACE: Uri=http://opcfoundation.org/UA/DI/"
"§NAMESPACE: Uri=http://br-automation.com/OpcUa/PLC/"
"§NAMESPACE: Uri=http://br-automation.com/OpcUa/PLC/PV/"

;Event 0 (TransitionEventType)
"§EVENT: TypeNs=0, TypeId=2311"
"§EVTFIELD: Name=/Message,						Var=::BrbUaSrvC:SrvTransitionEventData.Message"
"§EVTFIELD: Name=/Severity,						Var=::BrbUaSrvC:SrvTransitionEventData.nSeverity"
"§EVTFIELD: Name=/SourceName,					Var=::BrbUaSrvC:SrvTransitionEventData.sSourceName"
"§EVTFIELD: Name=/FromState,					Var=::BrbUaSrvC:SrvTransitionEventData.FromState"
"§EVTFIELD: Name=/FromState/Id,				Var=::BrbUaSrvC:SrvTransitionEventData.nFromStateId"
"§EVTFIELD: Name=/ToState,						Var=::BrbUaSrvC:SrvTransitionEventData.ToState"
"§EVTFIELD: Name=/ToState/Id,					Var=::BrbUaSrvC:SrvTransitionEventData.nToStateId"
"§EVTFIELD: Name=/Transition,					Var=::BrbUaSrvC:SrvTransitionEventData.Transition"
"§EVTFIELD: Name=/Transition/Id,			Var=::BrbUaSrvC:SrvTransitionEventData.nTransitionId"
```

### Program Logical/Tasks/BrbUa/BrbUaServer/BrbUaSrvC/BrbUaSrvC (ANSIC) - Server-Implementierung mit BrbLibUa in ANSI-C
